RoboDK station: Config_3_New_Drillbit.rdk

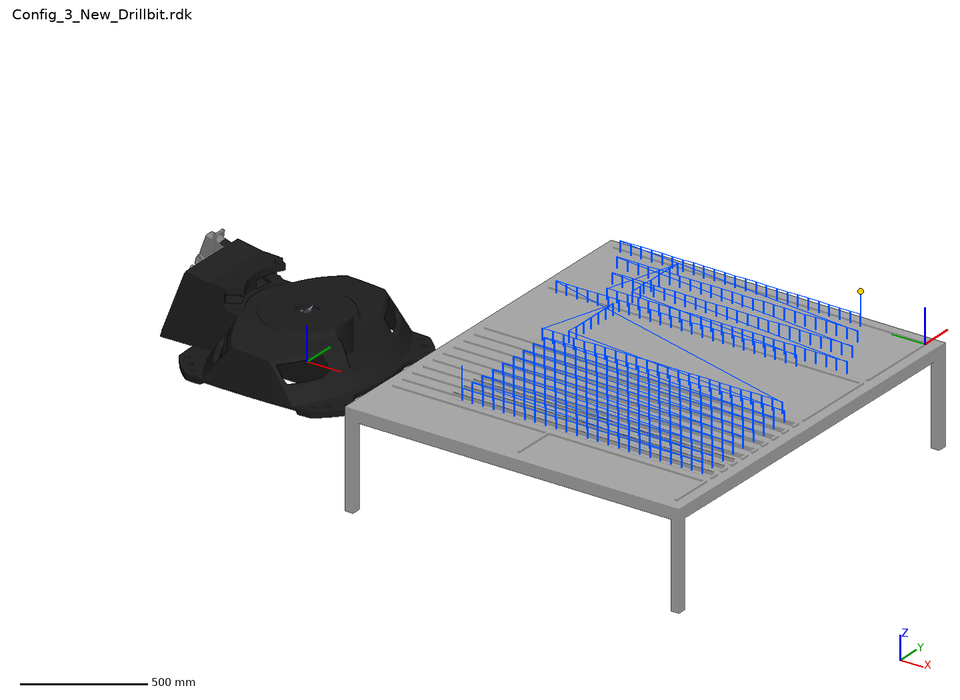
[picture v0: the station drawn from its stored meshes, robots at their saved joint values, targets as dots, program paths as lines]
Station Config_3_New_Drillbit (saved by RoboDK 5.2.3). Poses are relative to the parent item; angles as X-Y-Z fixed-axis rotations.
  - frame KUKA KR 210 R2700 extra Base at (0, 0, 0) mm
    - robot KUKA KR 210 R2700 extra: 6 axes, payload 210 kg, reach 2696 mm, repeatability 0.06 mm, weight 1068 kg
        joint limits [-185, -140, -120, -350, -125, -350] to [185, -5, 155, 350, 125, 350]; home [0, -90, 90, 0, 0, 0]; saved at [37.733, -88.827, 127.05, -51.844, 29.326, 78.997]
      - tool Spindle, TCP at (32, 0, 260) mm, rotated rx 0 ry 39 rz 0 deg, size 157.3 x 72 x 259.9 mm
  - frame Corner First Plate at (2495, 660, 510.8) mm, rotated rx 0 ry 0 rz 90 deg
  - object Table 3 at (1700, -800, 455) mm, rotated rx 0 ry 0 rz 90 deg, size 1820 x 1600 x 475 mm, geometry from Table 3.stl
  - object Config_3 at (2495, 660, 510.8) mm, rotated rx 0 ry 0 rz 90 deg
  - machining project Path1 settings: rotZ(0) | rotX(0)*rotY(0) | rotz(0) | onStart | onPathStart | onApproach | onPoint | onRetract | onFinish | SetRPM(%1) | SetTool(%1) | Extruder(%1) | default | default | OutOnMov(%1) | OutOffMov(%1) | onPathFinish | M_RunCode(%1)
  - program Path1 (1131 instructions, listed below)
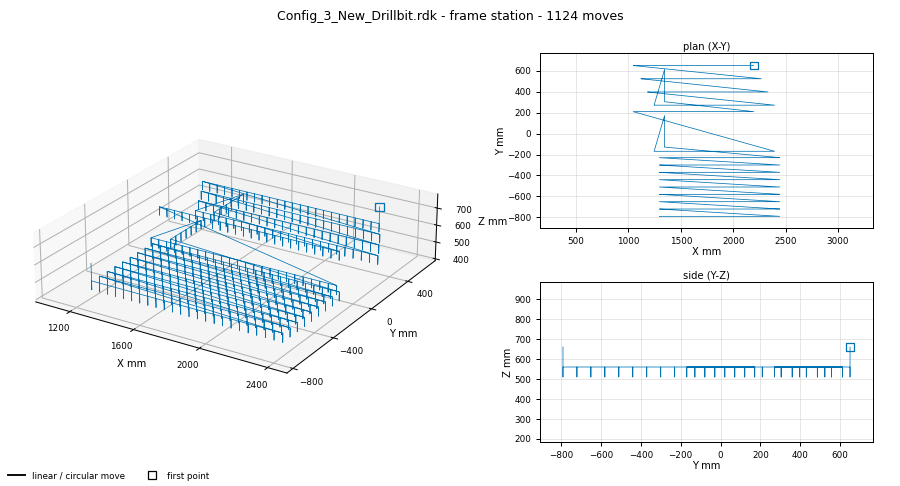
[picture p0: tool path of Config_3_New_Drillbit.rdk in frame station, 1124 of 1124 moves have a stored position in this frame; points joined in program order, loops and branches not executed]

--- program Path1 (robot KUKA KR 210 R2700 extra) ---
  Smooth(1)
  Set speed (1000.0 mm/s)
  Set Ref.: Corner First Plate
  Set Tool: Spindle
  Show Spindle
  MoveJ 1 to (-10.8, 300, 150) mm, rotated rx -180 ry 0 rz 90 deg; joints [-18.673, -56.771, 84.075, 25.785, 27.594, -37.894]
  MoveL 2 to (-10.8, 300, 150) mm, rotated rx -180 ry 0 rz 90 deg; joints [-18.673, -56.771, 84.075, 25.785, 27.594, -37.894]
  MoveL 3 to (-10.8, 300, 50) mm, rotated rx 180 ry 0 rz 90 deg; joints [-18.673, -54.184, 85.426, 29.563, 24.104, -42.09]
  MoveL 4 to (-10.8, 300, 50) mm, rotated rx 180 ry 0 rz 90 deg; joints [-18.673, -54.184, 85.426, 29.563, 24.104, -42.09]
  Set speed (150.0 mm/s)
  MoveL 5 to (-10.8, 300, -0.5) mm, rotated rx 180 ry 0 rz 90 deg; joints [-18.673, -52.769, 85.95, 31.865, 22.437, -44.595]
  MoveL 6 to (-10.8, 300, 50) mm, rotated rx 180 ry 0 rz 90 deg; joints [-18.673, -54.184, 85.426, 29.563, 24.104, -42.09]
  MoveL 7 to (-10.8, 350, 50) mm, rotated rx 180 ry 0 rz 90 deg; joints [-19.136, -56.141, 88.674, 31.59, 23.193, -44.569]
  MoveL 8 to (-10.8, 350, -0.5) mm, rotated rx 180 ry 0 rz 90 deg; joints [-19.136, -54.681, 89.197, 34.21, 21.527, -47.403]
  MoveL 9 to (-10.8, 350, 50) mm, rotated rx 180 ry 0 rz 90 deg; joints [-19.136, -56.141, 88.674, 31.59, 23.193, -44.569]
  MoveL 10 to (-10.8, 400, 50) mm, rotated rx -180 ry 0 rz 90 deg; joints [-19.622, -58.066, 91.821, 33.711, 22.382, -47.158]
  MoveL 11 to (-10.8, 400, -0.5) mm, rotated rx -180 ry 0 rz 90 deg; joints [-19.622, -56.557, 92.346, 36.679, 20.72, -50.348]
  MoveL 12 to (-10.8, 400, 50) mm, rotated rx -180 ry 0 rz 90 deg; joints [-19.622, -58.066, 91.821, 33.711, 22.382, -47.158]
  MoveL 13 to (-10.8, 450, 50) mm, rotated rx 180 ry 0 rz 90 deg; joints [-20.132, -59.962, 94.878, 35.915, 21.67, -49.846]
  MoveL 14 to (-10.8, 450, -0.5) mm, rotated rx -180 ry 0 rz 90 deg; joints [-20.132, -58.404, 95.405, 39.258, 20.016, -53.422]
  MoveL 15 to (-10.8, 450, 50) mm, rotated rx 180 ry 0 rz 90 deg; joints [-20.132, -59.962, 94.878, 35.915, 21.67, -49.846]
  MoveL 16 to (-10.8, 500, 50) mm, rotated rx 180 ry 0 rz 90 deg; joints [-20.668, -61.836, 97.851, 38.189, 21.056, -52.621]
  MoveL 17 to (-10.8, 500, -0.5) mm, rotated rx -180 ry 0 rz 90 deg; joints [-20.668, -60.227, 98.383, 41.928, 19.416, -56.606]
  MoveL 18 to (-10.8, 500, 50) mm, rotated rx 180 ry 0 rz 90 deg; joints [-20.668, -61.836, 97.851, 38.189, 21.056, -52.621]
  MoveL 19 to (-10.8, 550, 50) mm, rotated rx 180 ry 0 rz 90 deg; joints [-21.232, -63.693, 100.748, 40.512, 20.539, -55.465]
  MoveL 20 to (-10.8, 550, -0.5) mm, rotated rx -180 ry 0 rz 90 deg; joints [-21.232, -62.029, 101.285, 44.666, 18.917, -59.878]
  MoveL 21 to (-10.8, 550, 50) mm, rotated rx 180 ry 0 rz 90 deg; joints [-21.232, -63.693, 100.748, 40.512, 20.539, -55.465]
  MoveL 22 to (-10.8, 600, 50) mm, rotated rx -180 ry 0 rz 90 deg; joints [-21.826, -65.537, 103.573, 42.861, 20.119, -58.356]
  MoveL 23 to (-10.8, 600, -0.5) mm, rotated rx -180 ry 0 rz 90 deg; joints [-21.826, -63.817, 104.117, 47.441, 18.521, -63.209]
  MoveL 24 to (-10.8, 600, 50) mm, rotated rx -180 ry 0 rz 90 deg; joints [-21.826, -65.537, 103.573, 42.861, 20.119, -58.356]
  MoveL 25 to (-10.8, 650, 50) mm, rotated rx -180 ry 0 rz 90 deg; joints [-22.453, -67.372, 106.331, 45.208, 19.797, -61.269]
  MoveL 26 to (-10.8, 650, -0.5) mm, rotated rx 180 ry 0 rz 90 deg; joints [-22.453, -65.593, 106.883, 50.215, 18.227, -66.564]
  MoveL 27 to (-10.8, 650, 50) mm, rotated rx -180 ry 0 rz 90 deg; joints [-22.453, -67.372, 106.331, 45.208, 19.797, -61.269]
  MoveL 28 to (-10.8, 700, 50) mm, rotated rx -180 ry 0 rz 90 deg; joints [-23.115, -69.203, 109.025, 47.523, 19.571, -64.173]
  MoveL 29 to (-10.8, 700, -0.5) mm, rotated rx 180 ry 0 rz 90 deg; joints [-23.115, -67.362, 109.587, 52.95, 18.032, -69.905]
  MoveL 30 to (-10.8, 700, 50) mm, rotated rx -180 ry 0 rz 90 deg; joints [-23.115, -69.203, 109.025, 47.523, 19.571, -64.173]
  MoveL 31 to (-10.8, 750, 50) mm, rotated rx -180 ry 0 rz 90 deg; joints [-23.814, -71.033, 111.66, 49.773, 19.44, -67.039]
  MoveL 32 to (-10.8, 750, -0.5) mm, rotated rx 180 ry 0 rz 90 deg; joints [-23.814, -69.127, 112.233, 55.604, 17.936, -73.194]
  MoveL 33 to (-10.8, 750, 50) mm, rotated rx -180 ry 0 rz 90 deg; joints [-23.814, -71.033, 111.66, 49.773, 19.44, -67.039]
  MoveL 34 to (-10.8, 800, 50) mm, rotated rx -180 ry 0 rz 90 deg; joints [-24.555, -72.867, 114.238, 51.923, 19.404, -69.834]
  MoveL 35 to (-10.8, 800, -0.5) mm, rotated rx -180 ry 0 rz 90 deg; joints [-24.555, -70.893, 114.823, 58.134, 17.935, -76.388]
  MoveL 36 to (-10.8, 800, 50) mm, rotated rx -180 ry 0 rz 90 deg; joints [-24.555, -72.867, 114.238, 51.923, 19.404, -69.834]
  MoveL 37 to (-10.8, 850, 50) mm, rotated rx 180 ry 0 rz 90 deg; joints [-25.34, -74.708, 116.76, 53.942, 19.461, -72.529]
  MoveL 38 to (-10.8, 850, -0.5) mm, rotated rx -180 ry 0 rz 90 deg; joints [-25.34, -72.662, 117.358, 60.5, 18.027, -79.453]
  MoveL 39 to (-10.8, 850, 50) mm, rotated rx 180 ry 0 rz 90 deg; joints [-25.34, -74.708, 116.76, 53.942, 19.461, -72.529]
  MoveL 40 to (-10.8, 900, 50) mm, rotated rx -180 ry 0 rz 90 deg; joints [-26.173, -76.561, 119.228, 55.798, 19.61, -75.093]
  MoveL 41 to (-10.8, 900, -0.5) mm, rotated rx -180 ry 0 rz 90 deg; joints [-26.173, -74.439, 119.842, 62.666, 18.208, -82.352]
  MoveL 42 to (-10.8, 900, 50) mm, rotated rx -180 ry 0 rz 90 deg; joints [-26.173, -76.561, 119.228, 55.798, 19.61, -75.093]
  MoveL 43 to (-10.8, 950, 50) mm, rotated rx -180 ry 0 rz 90 deg; joints [-27.058, -78.43, 121.643, 57.462, 19.851, -77.502]
  MoveL 44 to (-10.8, 950, -0.5) mm, rotated rx 180 ry 0 rz 90 deg; joints [-27.058, -76.227, 122.274, 64.602, 18.476, -85.059]
  MoveL 45 to (-10.8, 950, 50) mm, rotated rx -180 ry 0 rz 90 deg; joints [-27.058, -78.43, 121.643, 57.462, 19.851, -77.502]
  MoveL 46 to (-10.8, 1000, 50) mm, rotated rx -180 ry 0 rz 90 deg; joints [-28.001, -80.318, 124.007, 58.912, 20.182, -79.735]
  MoveL 47 to (-10.8, 1000, -0.5) mm, rotated rx 180 ry 0 rz 90 deg; joints [-28.001, -78.031, 124.656, 66.28, 18.827, -87.549]
  MoveL 48 to (-10.8, 1000, 50) mm, rotated rx -180 ry 0 rz 90 deg; joints [-28.001, -80.318, 124.007, 58.912, 20.182, -79.735]
  MoveL 49 to (-10.8, 1050, 50) mm, rotated rx -180 ry 0 rz 90 deg; joints [-29.005, -82.231, 126.318, 60.129, 20.604, -81.776]
  MoveL 50 to (-10.8, 1050, -0.5) mm, rotated rx -180 ry 0 rz 90 deg; joints [-29.005, -79.854, 126.988, 67.681, 19.26, -89.808]
  MoveL 51 to (-10.8, 1050, 50) mm, rotated rx -180 ry 0 rz 90 deg; joints [-29.005, -82.231, 126.318, 60.129, 20.604, -81.776]
  MoveL 52 to (-10.8, 1100, 50) mm, rotated rx -180 ry 0 rz 90 deg; joints [-30.078, -84.172, 128.578, 61.097, 21.117, -83.613]
  MoveL 53 to (-10.8, 1100, -0.5) mm, rotated rx -180 ry 0 rz 90 deg; joints [-30.078, -81.701, 129.27, 68.792, 19.774, -91.823]
  MoveL 54 to (-10.8, 1100, 50) mm, rotated rx -180 ry 0 rz 90 deg; joints [-30.078, -84.172, 128.578, 61.097, 21.117, -83.613]
  MoveL 55 to (-10.8, 1150, 50) mm, rotated rx 180 ry 0 rz 90 deg; joints [-31.224, -86.147, 130.785, 61.808, 21.724, -85.24]
  MoveL 56 to (-10.8, 1150, -0.5) mm, rotated rx -180 ry 0 rz 90 deg; joints [-31.224, -83.576, 131.502, 69.603, 20.368, -93.59]
  MoveL 57 to (-10.8, 1150, 50) mm, rotated rx 180 ry 0 rz 90 deg; joints [-31.224, -86.147, 130.785, 61.808, 21.724, -85.24]
  MoveL 58 to (-10.8, 1200, 50) mm, rotated rx -180 ry 0 rz 90 deg; joints [-32.452, -88.16, 132.937, 62.257, 22.43, -86.657]
  MoveL 59 to (-10.8, 1200, -0.5) mm, rotated rx 180 ry 0 rz 90 deg; joints [-32.452, -85.485, 133.681, 70.11, 21.045, -95.109]
  MoveL 60 to (-10.8, 1200, 50) mm, rotated rx -180 ry 0 rz 90 deg; joints [-32.452, -88.16, 132.937, 62.257, 22.43, -86.657]
  MoveL 61 to (-10.8, 1250, 50) mm, rotated rx 180 ry 0 rz 90 deg; joints [-33.768, -90.216, 135.034, 62.444, 23.238, -87.866]
  MoveL 62 to (-10.8, 1250, -0.5) mm, rotated rx -180 ry 0 rz 90 deg; joints [-33.768, -87.431, 135.807, 70.315, 21.808, -96.384]
  MoveL 63 to (-10.8, 1250, 50) mm, rotated rx 180 ry 0 rz 90 deg; joints [-33.768, -90.216, 135.034, 62.444, 23.238, -87.866]
  MoveL 64 to (-10.8, 1300, 50) mm, rotated rx 180 ry 0 rz 90 deg; joints [-35.181, -92.32, 137.073, 62.376, 24.157, -88.879]
  MoveL 65 to (-10.8, 1300, -0.5) mm, rotated rx -180 ry 0 rz 90 deg; joints [-35.181, -89.419, 137.878, 70.222, 22.664, -97.425]
  MoveL 66 to (-10.8, 1300, 50) mm, rotated rx 180 ry 0 rz 90 deg; joints [-35.181, -92.32, 137.073, 62.376, 24.157, -88.879]
  MoveL 67 to (-10.8, 1350, 50) mm, rotated rx -180 ry 0 rz 90 deg; joints [-36.701, -94.476, 139.051, 62.061, 25.197, -89.708]
  MoveL 68 to (-10.8, 1350, -0.5) mm, rotated rx 180 ry 0 rz 90 deg; joints [-36.701, -91.455, 139.89, 69.839, 23.619, -98.245]
  MoveL 69 to (-10.8, 1350, 50) mm, rotated rx -180 ry 0 rz 90 deg; joints [-36.701, -94.476, 139.051, 62.061, 25.197, -89.708]
  MoveL 70 to (-10.8, 1400, 50) mm, rotated rx 180 ry 0 rz 90 deg; joints [-38.337, -96.689, 140.964, 61.514, 26.367, -90.372]
  MoveL 71 to (-10.8, 1400, -0.5) mm, rotated rx 180 ry 0 rz 90 deg; joints [-38.337, -93.543, 141.842, 69.179, 24.685, -98.863]
  MoveL 72 to (-10.8, 1400, 50) mm, rotated rx 180 ry 0 rz 90 deg; joints [-38.337, -96.689, 140.964, 61.514, 26.367, -90.372]
  MoveL 73 to (-10.8, 1450, 50) mm, rotated rx 180 ry 0 rz 90 deg; joints [-40.1, -98.961, 142.81, 60.755, 27.683, -90.897]
  MoveL 74 to (-10.8, 1450, -0.5) mm, rotated rx -180 ry 0 rz 90 deg; joints [-40.1, -95.687, 143.728, 68.26, 25.874, -99.3]
  MoveL 75 to (-10.8, 1450, 50) mm, rotated rx 180 ry 0 rz 90 deg; joints [-40.1, -98.961, 142.81, 60.755, 27.683, -90.897]
  MoveL 76 to (-136.94, 226.53, 50) mm, rotated rx -180 ry 0 rz 90 deg; joints [-14.696, -52.747, 83.017, 23.662, 23.44, -33.421]
  MoveL 77 to (-136.94, 226.53, -0.5) mm, rotated rx 180 ry 0 rz 90 deg; joints [-14.696, -51.366, 83.542, 25.573, 21.706, -35.49]
  MoveL 78 to (-136.94, 226.53, 50) mm, rotated rx -180 ry 0 rz 90 deg; joints [-14.696, -52.747, 83.017, 23.662, 23.44, -33.421]
  MoveL 79 to (-136.94, 276.53, 50) mm, rotated rx 180 ry 0 rz 90 deg; joints [-15.057, -54.772, 86.407, 25.489, 22.327, -35.605]
  MoveL 80 to (-136.94, 276.53, -0.5) mm, rotated rx -180 ry 0 rz 90 deg; joints [-15.057, -53.344, 86.931, 27.713, 20.582, -37.994]
  MoveL 81 to (-136.94, 276.53, 50) mm, rotated rx 180 ry 0 rz 90 deg; joints [-15.057, -54.772, 86.407, 25.489, 22.327, -35.605]
  MoveL 82 to (-136.94, 326.53, 50) mm, rotated rx 180 ry 0 rz 90 deg; joints [-15.435, -56.759, 89.689, 27.444, 21.31, -37.929]
  MoveL 83 to (-136.94, 326.53, -0.5) mm, rotated rx 180 ry 0 rz 90 deg; joints [-15.435, -55.284, 90.213, 30.025, 19.556, -40.683]
  MoveL 84 to (-136.94, 326.53, 50) mm, rotated rx 180 ry 0 rz 90 deg; joints [-15.435, -56.759, 89.689, 27.444, 21.31, -37.929]
  MoveL 85 to (-136.94, 376.53, 50) mm, rotated rx -180 ry 0 rz 90 deg; joints [-15.833, -58.716, 92.874, 29.528, 20.388, -40.394]
  MoveL 86 to (-136.94, 376.53, -0.5) mm, rotated rx 180 ry 0 rz 90 deg; joints [-15.833, -57.19, 93.4, 32.512, 18.63, -43.559]
  MoveL 87 to (-136.94, 376.53, 50) mm, rotated rx -180 ry 0 rz 90 deg; joints [-15.833, -58.716, 92.874, 29.528, 20.388, -40.394]
  MoveL 88 to (-136.94, 426.53, 50) mm, rotated rx 180 ry 0 rz 90 deg; joints [-16.251, -60.647, 95.97, 31.736, 19.561, -42.997]
  MoveL 89 to (-136.94, 426.53, -0.5) mm, rotated rx 180 ry 0 rz 90 deg; joints [-16.251, -59.071, 96.499, 35.17, 17.803, -46.621]
  MoveL 90 to (-136.94, 426.53, 50) mm, rotated rx 180 ry 0 rz 90 deg; joints [-16.251, -60.647, 95.97, 31.736, 19.561, -42.997]
  MoveL 91 to (-136.94, 476.53, 50) mm, rotated rx -180 ry 0 rz 90 deg; joints [-16.691, -62.56, 98.986, 34.06, 18.828, -45.731]
  MoveL 92 to (-136.94, 476.53, -0.5) mm, rotated rx -180 ry 0 rz 90 deg; joints [-16.691, -60.93, 99.52, 37.989, 17.077, -49.861]
  MoveL 93 to (-136.94, 476.53, 50) mm, rotated rx -180 ry 0 rz 90 deg; joints [-16.691, -62.56, 98.986, 34.06, 18.828, -45.731]
  MoveL 94 to (-136.94, 526.53, 50) mm, rotated rx 180 ry 0 rz 90 deg; joints [-17.155, -64.459, 101.928, 36.484, 18.191, -48.581]
  MoveL 95 to (-136.94, 526.53, -0.5) mm, rotated rx 180 ry 0 rz 90 deg; joints [-17.155, -62.773, 102.468, 40.951, 16.453, -53.259]
  MoveL 96 to (-136.94, 526.53, 50) mm, rotated rx 180 ry 0 rz 90 deg; joints [-17.155, -64.459, 101.928, 36.484, 18.191, -48.581]
  MoveL 97 to (-136.94, 576.53, 50) mm, rotated rx -180 ry 0 rz 90 deg; joints [-17.645, -66.35, 104.801, 38.987, 17.65, -51.528]
  MoveL 98 to (-136.94, 576.53, -0.5) mm, rotated rx 180 ry 0 rz 90 deg; joints [-17.645, -64.604, 105.349, 44.025, 15.931, -56.79]
  MoveL 99 to (-136.94, 576.53, 50) mm, rotated rx -180 ry 0 rz 90 deg; joints [-17.645, -66.35, 104.801, 38.987, 17.65, -51.528]
  MoveL 100 to (-136.94, 626.53, 50) mm, rotated rx -180 ry 0 rz 90 deg; joints [-18.163, -68.236, 107.61, 41.54, 17.206, -54.544]
  MoveL 101 to (-136.94, 626.53, -0.5) mm, rotated rx 180 ry 0 rz 90 deg; joints [-18.163, -66.429, 108.167, 47.173, 15.514, -60.415]
  MoveL 102 to (-136.94, 626.53, 50) mm, rotated rx -180 ry 0 rz 90 deg; joints [-18.163, -68.236, 107.61, 41.54, 17.206, -54.544]
  MoveL 103 to (-136.94, 676.53, 50) mm, rotated rx 180 ry 0 rz 90 deg; joints [-18.71, -70.124, 110.359, 44.108, 16.861, -57.597]
  MoveL 104 to (-136.94, 676.53, -0.5) mm, rotated rx 180 ry 0 rz 90 deg; joints [-18.71, -68.251, 110.926, 50.346, 15.201, -64.086]
  MoveL 105 to (-136.94, 676.53, 50) mm, rotated rx 180 ry 0 rz 90 deg; joints [-18.71, -70.124, 110.359, 44.108, 16.861, -57.597]
  MoveL 106 to (-136.94, 726.53, 50) mm, rotated rx -180 ry 0 rz 90 deg; joints [-19.291, -72.017, 113.051, 46.651, 16.613, -60.647]
  MoveL 107 to (-136.94, 726.53, -0.5) mm, rotated rx 180 ry 0 rz 90 deg; joints [-19.291, -70.075, 113.63, 53.486, 14.991, -67.75]
  MoveL 108 to (-136.94, 726.53, 50) mm, rotated rx -180 ry 0 rz 90 deg; joints [-19.291, -72.017, 113.051, 46.651, 16.613, -60.647]
  MoveL 109 to (-136.94, 776.53, 50) mm, rotated rx -180 ry 0 rz 90 deg; joints [-19.907, -73.921, 115.69, 49.122, 16.463, -63.65]
  MoveL 110 to (-136.94, 776.53, -0.5) mm, rotated rx -180 ry 0 rz 90 deg; joints [-19.907, -71.906, 116.282, 56.534, 14.884, -71.346]
  MoveL 111 to (-136.94, 776.53, 50) mm, rotated rx -180 ry 0 rz 90 deg; joints [-19.907, -73.921, 115.69, 49.122, 16.463, -63.65]
  MoveL 112 to (-136.94, 826.53, 50) mm, rotated rx -180 ry 0 rz 90 deg; joints [-20.562, -75.841, 118.277, 51.476, 16.411, -66.562]
  MoveL 113 to (-136.94, 826.53, -0.5) mm, rotated rx 180 ry 0 rz 90 deg; joints [-20.562, -73.748, 118.884, 59.426, 14.875, -74.816]
  MoveL 114 to (-136.94, 826.53, 50) mm, rotated rx -180 ry 0 rz 90 deg; joints [-20.562, -75.841, 118.277, 51.476, 16.411, -66.562]
  MoveL 115 to (-136.94, 876.53, 50) mm, rotated rx 180 ry 0 rz 90 deg; joints [-21.259, -77.781, 120.813, 53.664, 16.455, -69.337]
  MoveL 116 to (-136.94, 876.53, -0.5) mm, rotated rx 180 ry 0 rz 90 deg; joints [-21.259, -75.607, 121.438, 62.103, 14.963, -78.101]
  MoveL 117 to (-136.94, 876.53, 50) mm, rotated rx 180 ry 0 rz 90 deg; joints [-21.259, -77.781, 120.813, 53.664, 16.455, -69.337]
  MoveL 118 to (-136.94, 926.53, 50) mm, rotated rx 180 ry 0 rz 90 deg; joints [-22.003, -79.748, 123.302, 55.644, 16.595, -71.934]
  MoveL 119 to (-136.94, 926.53, -0.5) mm, rotated rx -180 ry 0 rz 90 deg; joints [-22.003, -77.487, 123.945, 64.512, 15.141, -81.151]
  MoveL 120 to (-136.94, 926.53, 50) mm, rotated rx 180 ry 0 rz 90 deg; joints [-22.003, -79.748, 123.302, 55.644, 16.595, -71.934]
  MoveL 121 to (-136.94, 976.53, 50) mm, rotated rx 180 ry 0 rz 90 deg; joints [-22.798, -81.747, 125.742, 57.374, 16.831, -74.315]
  MoveL 122 to (-136.94, 976.53, -0.5) mm, rotated rx 180 ry 0 rz 90 deg; joints [-22.798, -79.394, 126.407, 66.607, 15.408, -83.923]
  MoveL 123 to (-136.94, 976.53, 50) mm, rotated rx 180 ry 0 rz 90 deg; joints [-22.798, -81.747, 125.742, 57.374, 16.831, -74.315]
  MoveL 124 to (-136.94, 1026.53, 50) mm, rotated rx 180 ry 0 rz 90 deg; joints [-23.65, -83.786, 128.136, 58.822, 17.162, -76.449]
  MoveL 125 to (-136.94, 1026.53, -0.5) mm, rotated rx 180 ry 0 rz 90 deg; joints [-23.65, -81.334, 128.824, 68.353, 15.76, -86.384]
  MoveL 126 to (-136.94, 1026.53, 50) mm, rotated rx 180 ry 0 rz 90 deg; joints [-23.65, -83.786, 128.136, 58.822, 17.162, -76.449]
  MoveL 127 to (-136.94, 1076.53, 50) mm, rotated rx -180 ry 0 rz 90 deg; joints [-24.563, -85.871, 130.482, 59.961, 17.589, -78.313]
  MoveL 128 to (-136.94, 1076.53, -0.5) mm, rotated rx -180 ry 0 rz 90 deg; joints [-24.563, -83.315, 131.195, 69.722, 16.194, -88.511]
  MoveL 129 to (-136.94, 1076.53, 50) mm, rotated rx -180 ry 0 rz 90 deg; joints [-24.563, -85.871, 130.482, 59.961, 17.589, -78.313]
  MoveL 130 to (-136.94, 1126.53, 50) mm, rotated rx 180 ry 0 rz 90 deg; joints [-25.545, -88.01, 132.78, 60.772, 18.117, -79.89]
  MoveL 131 to (-136.94, 1126.53, -0.5) mm, rotated rx -180 ry 0 rz 90 deg; joints [-25.545, -85.343, 133.522, 70.696, 16.711, -90.288]
  MoveL 132 to (-136.94, 1126.53, 50) mm, rotated rx 180 ry 0 rz 90 deg; joints [-25.545, -88.01, 132.78, 60.772, 18.117, -79.89]
  MoveL 133 to (-136.94, 1176.53, 50) mm, rotated rx 180 ry 0 rz 90 deg; joints [-26.603, -90.212, 135.03, 61.243, 18.751, -81.173]
  MoveL 134 to (-136.94, 1176.53, -0.5) mm, rotated rx -180 ry 0 rz 90 deg; joints [-26.603, -87.427, 135.803, 71.264, 17.312, -91.708]
  MoveL 135 to (-136.94, 1176.53, 50) mm, rotated rx 180 ry 0 rz 90 deg; joints [-26.603, -90.212, 135.03, 61.243, 18.751, -81.173]
  MoveL 136 to (-136.94, 1226.53, 50) mm, rotated rx -180 ry 0 rz 90 deg; joints [-27.744, -92.486, 137.229, 61.372, 19.498, -82.16]
  MoveL 137 to (-136.94, 1226.53, -0.5) mm, rotated rx -180 ry 0 rz 90 deg; joints [-27.744, -89.576, 138.036, 71.423, 18.003, -92.77]
  MoveL 138 to (-136.94, 1226.53, 50) mm, rotated rx -180 ry 0 rz 90 deg; joints [-27.744, -92.486, 137.229, 61.372, 19.498, -82.16]
  MoveL 139 to (-136.94, 1276.53, 50) mm, rotated rx -180 ry 0 rz 90 deg; joints [-28.98, -94.842, 139.375, 61.162, 20.369, -82.86]
  MoveL 140 to (-136.94, 1276.53, -0.5) mm, rotated rx 180 ry 0 rz 90 deg; joints [-28.98, -91.801, 140.221, 71.174, 18.792, -93.483]
  MoveL 141 to (-136.94, 1276.53, 50) mm, rotated rx -180 ry 0 rz 90 deg; joints [-28.98, -94.842, 139.375, 61.162, 20.369, -82.86]
  MoveL 142 to (-136.94, 1326.53, 50) mm, rotated rx 180 ry 0 rz 90 deg; joints [-30.319, -97.292, 141.466, 60.624, 21.381, -83.287]
  MoveL 143 to (-136.94, 1326.53, -0.5) mm, rotated rx 180 ry 0 rz 90 deg; joints [-30.319, -94.113, 142.354, 70.527, 19.692, -93.857]
  MoveL 144 to (-136.94, 1326.53, 50) mm, rotated rx 180 ry 0 rz 90 deg; joints [-30.319, -97.292, 141.466, 60.624, 21.381, -83.287]
  MoveL 145 to (-136.94, 1376.53, 50) mm, rotated rx -180 ry 0 rz 90 deg; joints [-31.776, -99.848, 143.498, 59.78, 22.552, -83.466]
  MoveL 146 to (-136.94, 1376.53, -0.5) mm, rotated rx -180 ry 0 rz 90 deg; joints [-31.776, -96.524, 144.433, 69.496, 20.721, -93.913]
  MoveL 147 to (-136.94, 1376.53, 50) mm, rotated rx -180 ry 0 rz 90 deg; joints [-31.776, -99.848, 143.498, 59.78, 22.552, -83.466]
  MoveL 148 to (-263.08, 163.47, 50) mm, rotated rx -180 ry 0 rz 90 deg; joints [-10.919, -51.317, 80.596, 17.606, 23.211, -24.785]
  MoveL 149 to (-263.08, 163.47, -0.5) mm, rotated rx -180 ry 0 rz 90 deg; joints [-10.919, -49.967, 81.124, 19.044, 21.428, -26.34]
  MoveL 150 to (-263.08, 163.47, 50) mm, rotated rx -180 ry 0 rz 90 deg; joints [-10.919, -51.317, 80.596, 17.606, 23.211, -24.785]
  MoveL 151 to (-263.08, 213.47, 50) mm, rotated rx -180 ry 0 rz 90 deg; joints [-11.184, -53.402, 84.118, 19.086, 21.92, -26.532]
  MoveL 152 to (-263.08, 213.47, -0.5) mm, rotated rx 180 ry 0 rz 90 deg; joints [-11.184, -52.006, 84.643, 20.792, 20.113, -28.359]
  MoveL 153 to (-263.08, 213.47, 50) mm, rotated rx -180 ry 0 rz 90 deg; joints [-11.184, -53.402, 84.118, 19.086, 21.92, -26.532]
  MoveL 154 to (-263.08, 263.47, 50) mm, rotated rx -180 ry 0 rz 90 deg; joints [-11.463, -55.444, 87.522, 20.701, 20.719, -28.421]
  MoveL 155 to (-263.08, 263.47, -0.5) mm, rotated rx 180 ry 0 rz 90 deg; joints [-11.463, -54, 88.046, 22.723, 18.891, -30.569]
  MoveL 156 to (-263.08, 263.47, 50) mm, rotated rx -180 ry 0 rz 90 deg; joints [-11.463, -55.444, 87.522, 20.701, 20.719, -28.421]
  MoveL 157 to (-263.08, 313.47, 50) mm, rotated rx 180 ry 0 rz 90 deg; joints [-11.755, -57.451, 90.821, 22.46, 19.608, -30.463]
  MoveL 158 to (-263.08, 313.47, -0.5) mm, rotated rx -180 ry 0 rz 90 deg; joints [-11.755, -55.958, 91.346, 24.854, 17.76, -32.99]
  MoveL 159 to (-263.08, 313.47, 50) mm, rotated rx 180 ry 0 rz 90 deg; joints [-11.755, -57.451, 90.821, 22.46, 19.608, -30.463]
  MoveL 160 to (-263.08, 363.47, 50) mm, rotated rx -180 ry 0 rz 90 deg; joints [-12.062, -59.431, 94.026, 24.371, 18.585, -32.667]
  MoveL 161 to (-263.08, 363.47, -0.5) mm, rotated rx 180 ry 0 rz 90 deg; joints [-12.062, -57.887, 94.553, 27.202, 16.72, -35.637]
  MoveL 162 to (-263.08, 363.47, 50) mm, rotated rx -180 ry 0 rz 90 deg; joints [-12.062, -59.431, 94.026, 24.371, 18.585, -32.667]
  MoveL 163 to (-263.08, 413.47, 50) mm, rotated rx -180 ry 0 rz 90 deg; joints [-12.386, -61.389, 97.146, 26.438, 17.649, -35.037]
  MoveL 164 to (-263.08, 413.47, -0.5) mm, rotated rx 180 ry 0 rz 90 deg; joints [-12.386, -59.792, 97.676, 29.778, 15.771, -38.524]
  MoveL 165 to (-263.08, 413.47, 50) mm, rotated rx -180 ry 0 rz 90 deg; joints [-12.386, -61.389, 97.146, 26.438, 17.649, -35.037]
  MoveL 166 to (-263.08, 463.47, 50) mm, rotated rx 180 ry 0 rz 90 deg; joints [-12.727, -63.331, 100.187, 28.662, 16.801, -37.577]
  MoveL 167 to (-263.08, 463.47, -0.5) mm, rotated rx 180 ry 0 rz 90 deg; joints [-12.727, -61.678, 100.724, 32.588, 14.916, -41.658]
  MoveL 168 to (-263.08, 463.47, 50) mm, rotated rx 180 ry 0 rz 90 deg; joints [-12.727, -63.331, 100.187, 28.662, 16.801, -37.577]
  MoveL 169 to (-263.08, 513.47, 50) mm, rotated rx 180 ry 0 rz 90 deg; joints [-13.087, -65.264, 103.158, 31.038, 16.043, -40.283]
  MoveL 170 to (-263.08, 513.47, -0.5) mm, rotated rx 180 ry 0 rz 90 deg; joints [-13.087, -63.553, 103.701, 35.631, 14.158, -45.039]
  MoveL 171 to (-263.08, 513.47, 50) mm, rotated rx 180 ry 0 rz 90 deg; joints [-13.087, -65.264, 103.158, 31.038, 16.043, -40.283]
  MoveL 172 to (-263.08, 563.47, 50) mm, rotated rx -180 ry 0 rz 90 deg; joints [-13.467, -67.192, 106.063, 33.554, 15.377, -43.141]
  MoveL 173 to (-263.08, 563.47, -0.5) mm, rotated rx -180 ry 0 rz 90 deg; joints [-13.467, -65.419, 106.614, 38.891, 13.499, -48.652]
  MoveL 174 to (-263.08, 563.47, 50) mm, rotated rx -180 ry 0 rz 90 deg; joints [-13.467, -67.192, 106.063, 33.554, 15.377, -43.141]
  MoveL 175 to (-263.08, 613.47, 50) mm, rotated rx 180 ry 0 rz 90 deg; joints [-13.87, -69.121, 108.907, 36.187, 14.804, -46.133]
  MoveL 176 to (-263.08, 613.47, -0.5) mm, rotated rx 180 ry 0 rz 90 deg; joints [-13.87, -67.283, 109.468, 42.338, 12.944, -52.468]
  MoveL 177 to (-263.08, 613.47, 50) mm, rotated rx 180 ry 0 rz 90 deg; joints [-13.87, -69.121, 108.907, 36.187, 14.804, -46.133]
  MoveL 178 to (-263.08, 663.47, 50) mm, rotated rx -180 ry 0 rz 90 deg; joints [-14.297, -71.056, 111.693, 38.904, 14.328, -49.225]
  MoveL 179 to (-263.08, 663.47, -0.5) mm, rotated rx -180 ry 0 rz 90 deg; joints [-14.297, -69.15, 112.266, 45.923, 12.494, -56.44]
  MoveL 180 to (-263.08, 663.47, 50) mm, rotated rx -180 ry 0 rz 90 deg; joints [-14.297, -71.056, 111.693, 38.904, 14.328, -49.225]
  MoveL 181 to (-263.08, 713.47, 50) mm, rotated rx -180 ry 0 rz 90 deg; joints [-14.751, -73.003, 114.427, 41.662, 13.949, -52.376]
  MoveL 182 to (-263.08, 713.47, -0.5) mm, rotated rx 180 ry 0 rz 90 deg; joints [-14.751, -71.024, 115.012, 49.58, 12.15, -60.503]
  MoveL 183 to (-263.08, 713.47, 50) mm, rotated rx -180 ry 0 rz 90 deg; joints [-14.751, -73.003, 114.427, 41.662, 13.949, -52.376]
  MoveL 184 to (-263.08, 763.47, 50) mm, rotated rx -180 ry 0 rz 90 deg; joints [-15.234, -74.967, 117.109, 44.406, 13.67, -55.533]
  MoveL 185 to (-263.08, 763.47, -0.5) mm, rotated rx 180 ry 0 rz 90 deg; joints [-15.234, -72.911, 117.71, 53.225, 11.914, -64.575]
  MoveL 186 to (-263.08, 763.47, 50) mm, rotated rx -180 ry 0 rz 90 deg; joints [-15.234, -74.967, 117.109, 44.406, 13.67, -55.533]
  MoveL 187 to (-263.08, 813.47, 50) mm, rotated rx -180 ry 0 rz 90 deg; joints [-15.749, -76.955, 119.743, 47.073, 13.49, -58.634]
  MoveL 188 to (-263.08, 813.47, -0.5) mm, rotated rx -180 ry 0 rz 90 deg; joints [-15.749, -74.816, 120.361, 56.763, 11.784, -68.563]
  MoveL 189 to (-263.08, 813.47, 50) mm, rotated rx -180 ry 0 rz 90 deg; joints [-15.749, -76.955, 119.743, 47.073, 13.49, -58.634]
  MoveL 190 to (-263.08, 863.47, 50) mm, rotated rx 180 ry 0 rz 90 deg; joints [-16.299, -78.972, 122.331, 49.595, 13.411, -61.614]
  MoveL 191 to (-263.08, 863.47, -0.5) mm, rotated rx 180 ry 0 rz 90 deg; joints [-16.299, -76.746, 122.967, 60.097, 11.756, -72.371]
  MoveL 192 to (-263.08, 863.47, 50) mm, rotated rx 180 ry 0 rz 90 deg; joints [-16.299, -78.972, 122.331, 49.595, 13.411, -61.614]
  MoveL 193 to (-263.08, 913.47, 50) mm, rotated rx 180 ry 0 rz 90 deg; joints [-16.887, -81.027, 124.874, 51.903, 13.432, -64.404]
  MoveL 194 to (-263.08, 913.47, -0.5) mm, rotated rx -180 ry 0 rz 90 deg; joints [-16.887, -78.707, 125.531, 63.131, 11.826, -75.907]
  MoveL 195 to (-263.08, 913.47, 50) mm, rotated rx 180 ry 0 rz 90 deg; joints [-16.887, -81.027, 124.874, 51.903, 13.432, -64.404]
  MoveL 196 to (-263.08, 963.47, 50) mm, rotated rx 180 ry 0 rz 90 deg; joints [-17.518, -83.127, 127.373, 53.931, 13.554, -66.941]
  MoveL 197 to (-263.08, 963.47, -0.5) mm, rotated rx 180 ry 0 rz 90 deg; joints [-17.518, -80.708, 128.053, 65.783, 11.988, -79.089]
  MoveL 198 to (-263.08, 963.47, 50) mm, rotated rx 180 ry 0 rz 90 deg; joints [-17.518, -83.127, 127.373, 53.931, 13.554, -66.941]
  MoveL 199 to (-263.08, 1013.47, 50) mm, rotated rx 180 ry 0 rz 90 deg; joints [-18.197, -85.282, 129.829, 55.621, 13.776, -69.168]
  MoveL 200 to (-263.08, 1013.47, -0.5) mm, rotated rx 180 ry 0 rz 90 deg; joints [-18.197, -82.755, 130.535, 67.981, 12.239, -81.85]
  MoveL 201 to (-263.08, 1013.47, 50) mm, rotated rx 180 ry 0 rz 90 deg; joints [-18.197, -85.282, 129.829, 55.621, 13.776, -69.168]
  MoveL 202 to (-263.08, 1063.47, 50) mm, rotated rx 180 ry 0 rz 90 deg; joints [-18.928, -87.5, 132.242, 56.924, 14.1, -71.04]
  MoveL 203 to (-263.08, 1063.47, -0.5) mm, rotated rx -180 ry 0 rz 90 deg; joints [-18.928, -84.86, 132.977, 69.673, 12.574, -84.139]
  MoveL 204 to (-263.08, 1063.47, 50) mm, rotated rx 180 ry 0 rz 90 deg; joints [-18.928, -87.5, 132.242, 56.924, 14.1, -71.04]
  MoveL 205 to (-263.08, 1113.47, 50) mm, rotated rx -180 ry 0 rz 90 deg; joints [-19.718, -89.794, 134.612, 57.802, 14.532, -72.52]
  MoveL 206 to (-263.08, 1113.47, -0.5) mm, rotated rx 180 ry 0 rz 90 deg; joints [-19.718, -87.032, 135.379, 70.821, 12.991, -85.92]
  MoveL 207 to (-263.08, 1113.47, 50) mm, rotated rx -180 ry 0 rz 90 deg; joints [-19.718, -89.794, 134.612, 57.802, 14.532, -72.52]
  MoveL 208 to (-263.08, 1163.47, 50) mm, rotated rx 180 ry 0 rz 90 deg; joints [-20.574, -92.177, 136.938, 58.232, 15.077, -73.589]
  MoveL 209 to (-263.08, 1163.47, -0.5) mm, rotated rx 180 ry 0 rz 90 deg; joints [-20.574, -89.284, 137.74, 71.4, 13.494, -87.171]
  MoveL 210 to (-263.08, 1163.47, 50) mm, rotated rx 180 ry 0 rz 90 deg; joints [-20.574, -92.177, 136.938, 58.232, 15.077, -73.589]
  MoveL 211 to (-263.08, 1213.47, 50) mm, rotated rx -180 ry 0 rz 90 deg; joints [-21.503, -94.664, 139.218, 58.205, 15.748, -74.238]
  MoveL 212 to (-263.08, 1213.47, -0.5) mm, rotated rx 180 ry 0 rz 90 deg; joints [-21.503, -91.632, 140.06, 71.397, 14.087, -87.885]
  MoveL 213 to (-263.08, 1213.47, 50) mm, rotated rx -180 ry 0 rz 90 deg; joints [-21.503, -94.664, 139.218, 58.205, 15.748, -74.238]
  MoveL 214 to (-263.08, 1263.47, 50) mm, rotated rx 180 ry 0 rz 90 deg; joints [-22.516, -97.272, 141.45, 57.722, 16.562, -74.473]
  MoveL 215 to (-263.08, 1263.47, -0.5) mm, rotated rx 180 ry 0 rz 90 deg; joints [-22.516, -94.093, 142.337, 70.81, 14.784, -88.06]
  MoveL 216 to (-263.08, 1263.47, 50) mm, rotated rx 180 ry 0 rz 90 deg; joints [-22.516, -97.272, 141.45, 57.722, 16.562, -74.473]
  MoveL 217 to (-263.08, 1313.47, 50) mm, rotated rx -180 ry 0 rz 90 deg; joints [-23.624, -100.021, 143.63, 56.803, 17.54, -74.315]
  MoveL 218 to (-263.08, 1313.47, -0.5) mm, rotated rx -180 ry 0 rz 90 deg; joints [-23.624, -96.688, 144.568, 69.649, 15.604, -87.711]
  MoveL 219 to (-263.08, 1313.47, 50) mm, rotated rx -180 ry 0 rz 90 deg; joints [-23.624, -100.021, 143.63, 56.803, 17.54, -74.315]
  MoveL 220 to (-389.22, 100, 50) mm, rotated rx -180 ry 0 rz 90 deg; joints [-7.276, -49.461, 77.422, 11.443, 23.685, -16.168]
  MoveL 221 to (-389.22, 100, -0.5) mm, rotated rx -180 ry 0 rz 90 deg; joints [-7.276, -48.149, 77.954, 12.348, 21.881, -17.149]
  MoveL 222 to (-389.22, 100, 50) mm, rotated rx -180 ry 0 rz 90 deg; joints [-7.276, -49.461, 77.422, 11.443, 23.685, -16.168]
  MoveL 223 to (-389.22, 150, 50) mm, rotated rx 180 ry 0 rz 90 deg; joints [-7.449, -51.611, 81.094, 12.456, 22.228, -17.358]
  MoveL 224 to (-389.22, 150, -0.5) mm, rotated rx 180 ry 0 rz 90 deg; joints [-7.449, -50.254, 81.621, 13.542, 20.392, -18.524]
  MoveL 225 to (-389.22, 150, 50) mm, rotated rx 180 ry 0 rz 90 deg; joints [-7.449, -51.611, 81.094, 12.456, 22.228, -17.358]
  MoveL 226 to (-389.22, 200, 50) mm, rotated rx 180 ry 0 rz 90 deg; joints [-7.631, -53.71, 84.634, 13.574, 20.859, -18.659]
  MoveL 227 to (-389.22, 200, -0.5) mm, rotated rx 180 ry 0 rz 90 deg; joints [-7.631, -52.307, 85.158, 14.882, 18.991, -20.05]
  MoveL 228 to (-389.22, 200, 50) mm, rotated rx 180 ry 0 rz 90 deg; joints [-7.631, -53.71, 84.634, 13.574, 20.859, -18.659]
  MoveL 229 to (-389.22, 250, 50) mm, rotated rx 180 ry 0 rz 90 deg; joints [-7.823, -55.768, 88.058, 14.812, 19.575, -20.085]
  MoveL 230 to (-389.22, 250, -0.5) mm, rotated rx 180 ry 0 rz 90 deg; joints [-7.823, -54.316, 88.581, 16.389, 17.673, -21.748]
  MoveL 231 to (-389.22, 250, 50) mm, rotated rx 180 ry 0 rz 90 deg; joints [-7.823, -55.768, 88.058, 14.812, 19.575, -20.085]
  MoveL 232 to (-389.22, 300, 50) mm, rotated rx -180 ry 0 rz 90 deg; joints [-8.024, -57.793, 91.378, 16.182, 18.372, -21.649]
  MoveL 233 to (-389.22, 300, -0.5) mm, rotated rx 180 ry 0 rz 90 deg; joints [-8.024, -56.291, 91.902, 18.087, 16.436, -23.645]
  MoveL 234 to (-389.22, 300, 50) mm, rotated rx -180 ry 0 rz 90 deg; joints [-8.024, -57.793, 91.378, 16.182, 18.372, -21.649]
  MoveL 235 to (-389.22, 350, 50) mm, rotated rx 180 ry 0 rz 90 deg; joints [-8.235, -59.791, 94.605, 17.699, 17.248, -23.367]
  MoveL 236 to (-389.22, 350, -0.5) mm, rotated rx -180 ry 0 rz 90 deg; joints [-8.235, -58.238, 95.132, 20.004, 15.278, -25.768]
  MoveL 237 to (-389.22, 350, 50) mm, rotated rx 180 ry 0 rz 90 deg; joints [-8.235, -59.791, 94.605, 17.699, 17.248, -23.367]
  MoveL 238 to (-389.22, 400, 50) mm, rotated rx 180 ry 0 rz 90 deg; joints [-8.458, -61.771, 97.748, 19.375, 16.202, -25.252]
  MoveL 239 to (-389.22, 400, -0.5) mm, rotated rx 180 ry 0 rz 90 deg; joints [-8.458, -60.163, 98.28, 22.168, 14.201, -28.145]
  MoveL 240 to (-389.22, 400, 50) mm, rotated rx 180 ry 0 rz 90 deg; joints [-8.458, -61.771, 97.748, 19.375, 16.202, -25.252]
  MoveL 241 to (-389.22, 450, 50) mm, rotated rx -180 ry 0 rz 90 deg; joints [-8.693, -63.737, 100.815, 21.222, 15.234, -27.316]
  MoveL 242 to (-389.22, 450, -0.5) mm, rotated rx 180 ry 0 rz 90 deg; joints [-8.693, -62.072, 101.353, 24.607, 13.205, -30.807]
  MoveL 243 to (-389.22, 450, 50) mm, rotated rx -180 ry 0 rz 90 deg; joints [-8.693, -63.737, 100.815, 21.222, 15.234, -27.316]
  MoveL 244 to (-389.22, 500, 50) mm, rotated rx 180 ry 0 rz 90 deg; joints [-8.942, -65.695, 103.813, 23.25, 14.347, -29.571]
  MoveL 245 to (-389.22, 500, -0.5) mm, rotated rx -180 ry 0 rz 90 deg; joints [-8.942, -63.97, 104.358, 27.348, 12.294, -33.781]
  MoveL 246 to (-389.22, 500, 50) mm, rotated rx 180 ry 0 rz 90 deg; joints [-8.942, -65.695, 103.813, 23.25, 14.347, -29.571]
  MoveL 247 to (-389.22, 550, 50) mm, rotated rx 180 ry 0 rz 90 deg; joints [-9.205, -67.652, 106.747, 25.463, 13.542, -32.02]
  MoveL 248 to (-389.22, 550, -0.5) mm, rotated rx 180 ry 0 rz 90 deg; joints [-9.205, -65.864, 107.3, 30.411, 11.471, -37.087]
  MoveL 249 to (-389.22, 550, 50) mm, rotated rx 180 ry 0 rz 90 deg; joints [-9.205, -67.652, 106.747, 25.463, 13.542, -32.02]
  MoveL 250 to (-389.22, 600, 50) mm, rotated rx -180 ry 0 rz 90 deg; joints [-9.484, -69.613, 109.621, 27.857, 12.821, -34.66]
  MoveL 251 to (-389.22, 600, -0.5) mm, rotated rx 180 ry 0 rz 90 deg; joints [-9.484, -67.758, 110.185, 33.804, 10.741, -40.735]
  MoveL 252 to (-389.22, 600, 50) mm, rotated rx -180 ry 0 rz 90 deg; joints [-9.484, -69.613, 109.621, 27.857, 12.821, -34.66]
  MoveL 253 to (-389.22, 650, 50) mm, rotated rx 180 ry 0 rz 90 deg; joints [-9.78, -71.583, 112.44, 30.416, 12.19, -37.478]
  MoveL 254 to (-389.22, 650, -0.5) mm, rotated rx -180 ry 0 rz 90 deg; joints [-9.78, -69.657, 113.016, 37.514, 10.11, -44.711]
  MoveL 255 to (-389.22, 650, 50) mm, rotated rx 180 ry 0 rz 90 deg; joints [-9.78, -71.583, 112.44, 30.416, 12.19, -37.478]
  MoveL 256 to (-389.22, 700, 50) mm, rotated rx -180 ry 0 rz 90 deg; joints [-10.095, -73.57, 115.208, 33.111, 11.65, -40.445]
  MoveL 257 to (-389.22, 700, -0.5) mm, rotated rx -180 ry 0 rz 90 deg; joints [-10.095, -71.568, 115.798, 41.499, 9.583, -48.977]
  MoveL 258 to (-389.22, 700, 50) mm, rotated rx -180 ry 0 rz 90 deg; joints [-10.095, -73.57, 115.208, 33.111, 11.65, -40.445]
  MoveL 259 to (-389.22, 750, 50) mm, rotated rx -180 ry 0 rz 90 deg; joints [-10.431, -75.578, 117.928, 35.896, 11.205, -43.516]
  MoveL 260 to (-389.22, 750, -0.5) mm, rotated rx -180 ry 0 rz 90 deg; joints [-10.431, -73.497, 118.533, 45.682, 9.163, -53.456]
  MoveL 261 to (-389.22, 750, 50) mm, rotated rx -180 ry 0 rz 90 deg; joints [-10.431, -75.578, 117.928, 35.896, 11.205, -43.516]
  MoveL 262 to (-389.22, 800, 50) mm, rotated rx 180 ry 0 rz 90 deg; joints [-10.789, -77.616, 120.601, 38.705, 10.859, -46.625]
  MoveL 263 to (-389.22, 800, -0.5) mm, rotated rx -180 ry 0 rz 90 deg; joints [-10.789, -75.449, 121.225, 49.949, 8.853, -58.034]
  MoveL 264 to (-389.22, 800, 50) mm, rotated rx 180 ry 0 rz 90 deg; joints [-10.789, -77.616, 120.601, 38.705, 10.859, -46.625]
  MoveL 265 to (-389.22, 850, 50) mm, rotated rx -180 ry 0 rz 90 deg; joints [-11.173, -79.691, 123.231, 41.455, 10.614, -49.691]
  MoveL 266 to (-389.22, 850, -0.5) mm, rotated rx 180 ry 0 rz 90 deg; joints [-11.173, -77.432, 123.874, 54.149, 8.653, -62.564]
  MoveL 267 to (-389.22, 850, 50) mm, rotated rx -180 ry 0 rz 90 deg; joints [-11.173, -79.691, 123.231, 41.455, 10.614, -49.691]
  MoveL 268 to (-389.22, 900, 50) mm, rotated rx -180 ry 0 rz 90 deg; joints [-11.585, -81.811, 125.819, 44.048, 10.473, -52.619]
  MoveL 269 to (-389.22, 900, -0.5) mm, rotated rx 180 ry 0 rz 90 deg; joints [-11.585, -79.455, 126.484, 58.114, 8.559, -66.877]
  MoveL 270 to (-389.22, 900, 50) mm, rotated rx -180 ry 0 rz 90 deg; joints [-11.585, -81.811, 125.819, 44.048, 10.473, -52.619]
  MoveL 271 to (-389.22, 950, 50) mm, rotated rx 180 ry 0 rz 90 deg; joints [-12.027, -83.987, 128.366, 46.382, 10.436, -55.306]
  MoveL 272 to (-389.22, 950, -0.5) mm, rotated rx 180 ry 0 rz 90 deg; joints [-12.027, -81.525, 129.056, 61.672, 8.568, -70.804]
  MoveL 273 to (-389.22, 950, 50) mm, rotated rx 180 ry 0 rz 90 deg; joints [-12.027, -83.987, 128.366, 46.382, 10.436, -55.306]
  MoveL 274 to (-389.22, 1000, 50) mm, rotated rx 180 ry 0 rz 90 deg; joints [-12.505, -86.228, 130.873, 48.353, 10.507, -57.651]
  MoveL 275 to (-389.22, 1000, -0.5) mm, rotated rx -180 ry 0 rz 90 deg; joints [-12.505, -83.653, 131.591, 64.668, 8.671, -74.192]
  MoveL 276 to (-389.22, 1000, 50) mm, rotated rx 180 ry 0 rz 90 deg; joints [-12.505, -86.228, 130.873, 48.353, 10.507, -57.651]
  MoveL 277 to (-389.22, 1050, 50) mm, rotated rx 180 ry 0 rz 90 deg; joints [-13.021, -88.548, 133.341, 49.869, 10.687, -59.563]
  MoveL 278 to (-389.22, 1050, -0.5) mm, rotated rx -180 ry 0 rz 90 deg; joints [-13.021, -85.852, 134.09, 66.974, 8.862, -76.913]
  MoveL 279 to (-389.22, 1050, 50) mm, rotated rx 180 ry 0 rz 90 deg; joints [-13.021, -88.548, 133.341, 49.869, 10.687, -59.563]
  MoveL 280 to (-389.22, 1100, 50) mm, rotated rx 180 ry 0 rz 90 deg; joints [-13.58, -90.962, 135.769, 50.857, 10.984, -60.97]
  MoveL 281 to (-389.22, 1100, -0.5) mm, rotated rx -180 ry 0 rz 90 deg; joints [-13.58, -88.136, 136.553, 68.495, 9.139, -78.876]
  MoveL 282 to (-389.22, 1100, 50) mm, rotated rx 180 ry 0 rz 90 deg; joints [-13.58, -90.962, 135.769, 50.857, 10.984, -60.97]
  MoveL 283 to (-389.22, 1150, 50) mm, rotated rx 180 ry 0 rz 90 deg; joints [-14.189, -93.486, 138.156, 51.264, 11.406, -61.822]
  MoveL 284 to (-389.22, 1150, -0.5) mm, rotated rx 180 ry 0 rz 90 deg; joints [-14.189, -90.521, 138.98, 69.167, 9.5, -80.019]
  MoveL 285 to (-389.22, 1150, 50) mm, rotated rx 180 ry 0 rz 90 deg; joints [-14.189, -93.486, 138.156, 51.264, 11.406, -61.822]
  MoveL 286 to (-389.22, 1200, 50) mm, rotated rx -180 ry 0 rz 90 deg; joints [-14.854, -96.142, 140.502, 51.068, 11.97, -62.098]
  MoveL 287 to (-389.22, 1200, -0.5) mm, rotated rx 180 ry 0 rz 90 deg; joints [-14.854, -93.027, 141.37, 68.955, 9.954, -80.309]
  MoveL 288 to (-389.22, 1200, 50) mm, rotated rx -180 ry 0 rz 90 deg; joints [-14.854, -96.142, 140.502, 51.068, 11.97, -62.098]
  MoveL 289 to (-389.22, 1250, 50) mm, rotated rx -180 ry 0 rz 90 deg; joints [-15.583, -98.954, 142.804, 50.274, 12.698, -61.804]
  MoveL 290 to (-389.22, 1250, -0.5) mm, rotated rx -180 ry 0 rz 90 deg; joints [-15.583, -95.68, 143.722, 67.852, 10.517, -79.74]
  MoveL 291 to (-389.22, 1250, 50) mm, rotated rx -180 ry 0 rz 90 deg; joints [-15.583, -98.954, 142.804, 50.274, 12.698, -61.804]
  MoveL 292 to (-48.6, 1150, 50) mm, rotated rx -180 ry 0 rz 90 deg; joints [-29.722, -87.047, 131.759, 61.733, 20.748, -84.027]
  MoveL 293 to (-48.6, 1150, -0.5) mm, rotated rx 180 ry 0 rz 90 deg; joints [-29.722, -84.43, 132.488, 70.106, 19.379, -92.938]
  MoveL 294 to (-48.6, 1150, 50) mm, rotated rx -180 ry 0 rz 90 deg; joints [-29.722, -87.047, 131.759, 61.733, 20.748, -84.027]
  MoveL 295 to (-103.93, 1150, 50) mm, rotated rx -180 ry 0 rz 90 deg; joints [-27.44, -88.313, 133.097, 61.393, 19.289, -81.956]
  MoveL 296 to (-103.93, 1150, -0.5) mm, rotated rx 180 ry 0 rz 90 deg; joints [-27.44, -85.63, 133.842, 70.725, 17.892, -91.798]
  MoveL 297 to (-103.93, 1150, 50) mm, rotated rx -180 ry 0 rz 90 deg; joints [-27.44, -88.313, 133.097, 61.393, 19.289, -81.956]
  MoveL 298 to (-174.73, 1150, 50) mm, rotated rx 180 ry 0 rz 90 deg; joints [-24.376, -89.829, 134.647, 60.454, 17.371, -78.692]
  MoveL 299 to (-174.73, 1150, -0.5) mm, rotated rx -180 ry 0 rz 90 deg; joints [-24.376, -87.064, 135.414, 71.253, 15.92, -89.959]
  MoveL 300 to (-174.73, 1150, 50) mm, rotated rx 180 ry 0 rz 90 deg; joints [-24.376, -89.829, 134.647, 60.454, 17.371, -78.692]
  MoveL 301 to (-230.06, 1150, 50) mm, rotated rx 180 ry 0 rz 90 deg; joints [-21.873, -90.919, 135.727, 59.196, 15.841, -75.539]
  MoveL 302 to (-230.06, 1150, -0.5) mm, rotated rx 180 ry 0 rz 90 deg; joints [-21.873, -88.096, 136.511, 71.382, 14.324, -88.155]
  MoveL 303 to (-230.06, 1150, 50) mm, rotated rx 180 ry 0 rz 90 deg; joints [-21.873, -90.919, 135.727, 59.196, 15.841, -75.539]
  MoveL 304 to (-300.86, 1150, 50) mm, rotated rx 180 ry 0 rz 90 deg; joints [-18.539, -92.175, 136.935, 56.652, 13.859, -70.477]
  MoveL 305 to (-300.86, 1150, -0.5) mm, rotated rx -180 ry 0 rz 90 deg; joints [-18.539, -89.282, 137.738, 71.018, 12.216, -85.218]
  MoveL 306 to (-300.86, 1150, 50) mm, rotated rx 180 ry 0 rz 90 deg; joints [-18.539, -92.175, 136.935, 56.652, 13.859, -70.477]
  MoveL 307 to (-356.19, 1150, 50) mm, rotated rx -180 ry 0 rz 90 deg; joints [-15.838, -93.032, 137.738, 53.642, 12.314, -65.436]
  MoveL 308 to (-356.19, 1150, -0.5) mm, rotated rx 180 ry 0 rz 90 deg; joints [-15.838, -90.092, 138.554, 70.106, 10.524, -82.226]
  MoveL 309 to (-356.19, 1150, 50) mm, rotated rx -180 ry 0 rz 90 deg; joints [-15.838, -93.032, 137.738, 53.642, 12.314, -65.436]
  MoveL 310 to (-450.8, 300, 50) mm, rotated rx -180 ry 0 rz 90 deg; joints [-6.215, -58.102, 91.881, 12.873, 17.807, -17.113]
  MoveL 311 to (-450.8, 300, -0.5) mm, rotated rx 180 ry 0 rz 90 deg; joints [-6.215, -56.593, 92.406, 14.464, 15.83, -18.775]
  MoveL 312 to (-450.8, 300, 50) mm, rotated rx -180 ry 0 rz 90 deg; joints [-6.215, -58.102, 91.881, 12.873, 17.807, -17.113]
  MoveL 313 to (-450.8, 350, 50) mm, rotated rx 180 ry 0 rz 90 deg; joints [-6.38, -60.106, 95.108, 14.128, 16.649, -18.524]
  MoveL 314 to (-450.8, 350, -0.5) mm, rotated rx -180 ry 0 rz 90 deg; joints [-6.38, -58.544, 95.636, 16.073, 14.631, -20.543]
  MoveL 315 to (-450.8, 350, 50) mm, rotated rx 180 ry 0 rz 90 deg; joints [-6.38, -60.106, 95.108, 14.128, 16.649, -18.524]
  MoveL 316 to (-450.8, 400, 50) mm, rotated rx 180 ry 0 rz 90 deg; joints [-6.554, -62.091, 98.252, 15.527, 15.565, -20.085]
  MoveL 317 to (-450.8, 400, -0.5) mm, rotated rx 180 ry 0 rz 90 deg; joints [-6.554, -60.474, 98.784, 17.912, 13.506, -22.549]
  MoveL 318 to (-450.8, 400, 50) mm, rotated rx 180 ry 0 rz 90 deg; joints [-6.554, -62.091, 98.252, 15.527, 15.565, -20.085]
  MoveL 319 to (-450.8, 450, 50) mm, rotated rx 180 ry 0 rz 90 deg; joints [-6.737, -64.065, 101.321, 17.085, 14.554, -21.813]
  MoveL 320 to (-450.8, 450, -0.5) mm, rotated rx 180 ry 0 rz 90 deg; joints [-6.737, -62.39, 101.86, 20.018, 12.455, -24.828]
  MoveL 321 to (-450.8, 450, 50) mm, rotated rx 180 ry 0 rz 90 deg; joints [-6.737, -64.065, 101.321, 17.085, 14.554, -21.813]
  MoveL 322 to (-450.8, 500, 50) mm, rotated rx -180 ry 0 rz 90 deg; joints [-6.931, -66.032, 104.322, 18.817, 13.618, -23.721]
  MoveL 323 to (-450.8, 500, -0.5) mm, rotated rx 180 ry 0 rz 90 deg; joints [-6.931, -64.297, 104.869, 22.428, 11.481, -27.42]
  MoveL 324 to (-450.8, 500, 50) mm, rotated rx -180 ry 0 rz 90 deg; joints [-6.931, -66.032, 104.322, 18.817, 13.618, -23.721]
  MoveL 325 to (-450.8, 550, 50) mm, rotated rx 180 ry 0 rz 90 deg; joints [-7.136, -67.999, 107.26, 20.733, 12.758, -25.821]
  MoveL 326 to (-450.8, 550, -0.5) mm, rotated rx -180 ry 0 rz 90 deg; joints [-7.136, -66.2, 107.816, 25.181, 10.588, -30.361]
  MoveL 327 to (-450.8, 550, 50) mm, rotated rx 180 ry 0 rz 90 deg; joints [-7.136, -67.999, 107.26, 20.733, 12.758, -25.821]
  MoveL 328 to (-450.8, 600, 50) mm, rotated rx 180 ry 0 rz 90 deg; joints [-7.354, -69.972, 110.14, 22.839, 11.978, -28.119]
  MoveL 329 to (-450.8, 600, -0.5) mm, rotated rx -180 ry 0 rz 90 deg; joints [-7.354, -68.105, 110.707, 28.308, 9.78, -33.687]
  MoveL 330 to (-450.8, 600, 50) mm, rotated rx 180 ry 0 rz 90 deg; joints [-7.354, -69.972, 110.14, 22.839, 11.978, -28.119]
  MoveL 331 to (-450.8, 650, 50) mm, rotated rx -180 ry 0 rz 90 deg; joints [-7.585, -71.957, 112.966, 25.131, 11.28, -30.612]
  MoveL 332 to (-450.8, 650, -0.5) mm, rotated rx 180 ry 0 rz 90 deg; joints [-7.585, -70.017, 113.545, 31.829, 9.063, -37.416]
  MoveL 333 to (-450.8, 650, 50) mm, rotated rx -180 ry 0 rz 90 deg; joints [-7.585, -71.957, 112.966, 25.131, 11.28, -30.612]
  MoveL 334 to (-450.8, 700, 50) mm, rotated rx 180 ry 0 rz 90 deg; joints [-7.832, -73.959, 115.742, 27.592, 10.67, -33.285]
  MoveL 335 to (-450.8, 700, -0.5) mm, rotated rx -180 ry 0 rz 90 deg; joints [-7.832, -71.943, 116.335, 35.736, 8.443, -41.542]
  MoveL 336 to (-450.8, 700, 50) mm, rotated rx 180 ry 0 rz 90 deg; joints [-7.832, -73.959, 115.742, 27.592, 10.67, -33.285]
  MoveL 337 to (-450.8, 750, 50) mm, rotated rx -180 ry 0 rz 90 deg; joints [-8.094, -75.987, 118.47, 30.188, 10.15, -36.103]
  MoveL 338 to (-450.8, 750, -0.5) mm, rotated rx -180 ry 0 rz 90 deg; joints [-8.094, -73.888, 119.079, 39.985, 7.926, -46.022]
  MoveL 339 to (-450.8, 750, 50) mm, rotated rx -180 ry 0 rz 90 deg; joints [-8.094, -75.987, 118.47, 30.188, 10.15, -36.103]
  MoveL 340 to (-450.8, 800, 50) mm, rotated rx -180 ry 0 rz 90 deg; joints [-8.375, -78.046, 121.154, 32.862, 9.726, -39.012]
  MoveL 341 to (-450.8, 800, -0.5) mm, rotated rx 180 ry 0 rz 90 deg; joints [-8.375, -75.86, 121.781, 44.477, 7.518, -50.757]
  MoveL 342 to (-450.8, 800, 50) mm, rotated rx -180 ry 0 rz 90 deg; joints [-8.375, -78.046, 121.154, 32.862, 9.726, -39.012]
  MoveL 343 to (-450.8, 850, 50) mm, rotated rx 180 ry 0 rz 90 deg; joints [-8.676, -80.146, 123.795, 35.535, 9.401, -41.932]
  MoveL 344 to (-450.8, 850, -0.5) mm, rotated rx -180 ry 0 rz 90 deg; joints [-8.676, -77.867, 124.442, 49.054, 7.22, -55.591]
  MoveL 345 to (-450.8, 850, 50) mm, rotated rx 180 ry 0 rz 90 deg; joints [-8.676, -80.146, 123.795, 35.535, 9.401, -41.932]
  MoveL 346 to (-450.8, 900, 50) mm, rotated rx 180 ry 0 rz 90 deg; joints [-8.999, -82.295, 126.395, 38.103, 9.179, -44.761]
  MoveL 347 to (-450.8, 900, -0.5) mm, rotated rx 180 ry 0 rz 90 deg; joints [-8.999, -79.915, 127.066, 53.508, 7.033, -60.317]
  MoveL 348 to (-450.8, 900, 50) mm, rotated rx 180 ry 0 rz 90 deg; joints [-8.999, -82.295, 126.395, 38.103, 9.179, -44.761]
  MoveL 349 to (-450.8, 950, 50) mm, rotated rx -180 ry 0 rz 90 deg; joints [-9.347, -84.504, 128.955, 40.447, 9.065, -47.382]
  MoveL 350 to (-450.8, 950, -0.5) mm, rotated rx -180 ry 0 rz 90 deg; joints [-9.347, -82.017, 129.652, 57.6, 6.953, -64.698]
  MoveL 351 to (-450.8, 950, 50) mm, rotated rx -180 ry 0 rz 90 deg; joints [-9.347, -84.504, 128.955, 40.447, 9.065, -47.382]
  MoveL 352 to (-450.8, 1000, 50) mm, rotated rx 180 ry 0 rz 90 deg; joints [-9.723, -86.785, 131.477, 42.441, 9.061, -49.668]
  MoveL 353 to (-450.8, 1000, -0.5) mm, rotated rx -180 ry 0 rz 90 deg; joints [-9.723, -84.181, 132.203, 61.093, 6.973, -68.497]
  MoveL 354 to (-450.8, 1000, 50) mm, rotated rx 180 ry 0 rz 90 deg; joints [-9.723, -86.785, 131.477, 42.441, 9.061, -49.668]
  MoveL 355 to (-450.8, 1050, 50) mm, rotated rx 180 ry 0 rz 90 deg; joints [-10.13, -89.151, 133.961, 43.967, 9.174, -51.503]
  MoveL 356 to (-450.8, 1050, -0.5) mm, rotated rx -180 ry 0 rz 90 deg; joints [-10.13, -86.423, 134.719, 63.779, 7.087, -71.509]
  MoveL 357 to (-450.8, 1050, 50) mm, rotated rx 180 ry 0 rz 90 deg; joints [-10.13, -89.151, 133.961, 43.967, 9.174, -51.503]
  MoveL 358 to (-450.8, 1100, 50) mm, rotated rx -180 ry 0 rz 90 deg; joints [-10.571, -91.62, 136.406, 44.925, 9.41, -52.789]
  MoveL 359 to (-450.8, 1100, -0.5) mm, rotated rx 180 ry 0 rz 90 deg; joints [-10.571, -88.758, 137.2, 65.501, 7.289, -73.577]
  MoveL 360 to (-450.8, 1100, 50) mm, rotated rx -180 ry 0 rz 90 deg; joints [-10.571, -91.62, 136.406, 44.925, 9.41, -52.789]
  MoveL 361 to (-450.8, 1150, 50) mm, rotated rx -180 ry 0 rz 90 deg; joints [-11.053, -94.21, 138.812, 45.246, 9.782, -53.459]
  MoveL 362 to (-450.8, 1150, -0.5) mm, rotated rx -180 ry 0 rz 90 deg; joints [-11.053, -91.204, 139.648, 66.152, 7.58, -74.597]
  MoveL 363 to (-450.8, 1150, 50) mm, rotated rx -180 ry 0 rz 90 deg; joints [-11.053, -94.21, 138.812, 45.246, 9.782, -53.459]
  MoveL 364 to (-450.8, 1200, 50) mm, rotated rx -180 ry 0 rz 90 deg; joints [-11.58, -96.945, 141.178, 44.903, 10.309, -53.485]
  MoveL 365 to (-450.8, 1200, -0.5) mm, rotated rx -180 ry 0 rz 90 deg; joints [-11.58, -93.785, 142.06, 65.678, 7.969, -74.517]
  MoveL 366 to (-450.8, 1200, 50) mm, rotated rx -180 ry 0 rz 90 deg; joints [-11.58, -96.945, 141.178, 44.903, 10.309, -53.485]
  MoveL 367 to (-450.8, 1250, 50) mm, rotated rx -180 ry 0 rz 90 deg; joints [-12.159, -99.852, 143.501, 43.912, 11.018, -52.885]
  MoveL 368 to (-450.8, 1250, -0.5) mm, rotated rx -180 ry 0 rz 90 deg; joints [-12.159, -96.528, 144.436, 64.079, 8.475, -73.337]
  MoveL 369 to (-450.8, 1250, 50) mm, rotated rx -180 ry 0 rz 90 deg; joints [-12.159, -99.852, 143.501, 43.912, 11.018, -52.885]
  MoveL 370 to (-450.8, 1300, 50) mm, rotated rx -180 ry 0 rz 90 deg; joints [-12.798, -102.966, 145.779, 42.33, 11.948, -51.718]
  MoveL 371 to (-450.8, 1300, -0.5) mm, rotated rx -180 ry 0 rz 90 deg; joints [-12.798, -99.47, 146.773, 61.412, 9.135, -71.116]
  MoveL 372 to (-450.8, 1300, 50) mm, rotated rx -180 ry 0 rz 90 deg; joints [-12.798, -102.966, 145.779, 42.33, 11.948, -51.718]
  MoveL 373 to (-450.8, 1350, 50) mm, rotated rx -180 ry 0 rz 90 deg; joints [-13.507, -106.329, 148.005, 40.257, 13.147, -50.082]
  MoveL 374 to (-450.8, 1350, -0.5) mm, rotated rx -180 ry 0 rz 90 deg; joints [-13.507, -102.653, 149.068, 57.804, 10.002, -67.98]
  MoveL 375 to (-450.8, 1350, 50) mm, rotated rx -180 ry 0 rz 90 deg; joints [-13.507, -106.329, 148.005, 40.257, 13.147, -50.082]
  MoveL 376 to (-450.8, 1400, 50) mm, rotated rx 180 ry 0 rz 90 deg; joints [-14.296, -109.989, 150.175, 37.819, 14.681, -48.104]
  MoveL 377 to (-450.8, 1400, -0.5) mm, rotated rx -180 ry 0 rz 90 deg; joints [-14.296, -106.134, 151.316, 53.454, 11.153, -64.132]
  MoveL 378 to (-450.8, 1400, 50) mm, rotated rx 180 ry 0 rz 90 deg; joints [-14.296, -109.989, 150.175, 37.819, 14.681, -48.104]
  MoveL 379 to (-450.8, 1450, 50) mm, rotated rx 180 ry 0 rz 90 deg; joints [-15.182, -114.009, 152.278, 35.161, 16.63, -45.925]
  MoveL 380 to (-450.8, 1450, -0.5) mm, rotated rx 180 ry 0 rz 90 deg; joints [-15.182, -109.981, 153.51, 48.629, 12.687, -59.834]
  MoveL 381 to (-450.8, 1450, 50) mm, rotated rx 180 ry 0 rz 90 deg; joints [-15.182, -114.009, 152.278, 35.161, 16.63, -45.925]
  MoveL 382 to (-829.2, 100, 50) mm, rotated rx 180 ry 0 rz 90 deg; joints [4.561, -49.92, 78.21, -7.368, 22.969, 10.337]
  MoveL 383 to (-829.2, 100, -0.5) mm, rotated rx 180 ry 0 rz 90 deg; joints [4.561, -48.599, 78.741, -7.979, 21.134, 10.996]
  MoveL 384 to (-829.2, 100, 50) mm, rotated rx 180 ry 0 rz 90 deg; joints [4.561, -49.92, 78.21, -7.368, 22.969, 10.337]
  MoveL 385 to (-829.2, 150, 50) mm, rotated rx 180 ry 0 rz 90 deg; joints [4.671, -52.069, 81.871, -8.044, 21.484, 11.124]
  MoveL 386 to (-829.2, 150, -0.5) mm, rotated rx 180 ry 0 rz 90 deg; joints [4.671, -50.702, 82.397, -8.783, 19.611, 11.913]
  MoveL 387 to (-829.2, 150, 50) mm, rotated rx 180 ry 0 rz 90 deg; joints [4.671, -52.069, 81.871, -8.044, 21.484, 11.124]
  MoveL 388 to (-829.2, 200, 50) mm, rotated rx 180 ry 0 rz 90 deg; joints [4.786, -54.17, 85.403, -8.796, 20.082, 11.991]
  MoveL 389 to (-829.2, 200, -0.5) mm, rotated rx 180 ry 0 rz 90 deg; joints [4.786, -52.756, 85.927, -9.694, 18.169, 12.941]
  MoveL 390 to (-829.2, 200, 50) mm, rotated rx 180 ry 0 rz 90 deg; joints [4.786, -54.17, 85.403, -8.796, 20.082, 11.991]
  MoveL 391 to (-829.2, 250, 50) mm, rotated rx 180 ry 0 rz 90 deg; joints [4.907, -56.231, 88.821, -9.635, 18.759, 12.949]
  MoveL 392 to (-829.2, 250, -0.5) mm, rotated rx -180 ry 0 rz 90 deg; joints [4.907, -54.768, 89.345, -10.731, 16.804, 14.099]
  MoveL 393 to (-829.2, 250, 50) mm, rotated rx 180 ry 0 rz 90 deg; joints [4.907, -56.231, 88.821, -9.635, 18.759, 12.949]
  MoveL 394 to (-829.2, 300, 50) mm, rotated rx -180 ry 0 rz 90 deg; joints [5.034, -58.261, 92.139, -10.575, 17.51, 14.011]
  MoveL 395 to (-829.2, 300, -0.5) mm, rotated rx 180 ry 0 rz 90 deg; joints [5.034, -56.748, 92.664, -11.916, 15.511, 15.41]
  MoveL 396 to (-829.2, 300, 50) mm, rotated rx -180 ry 0 rz 90 deg; joints [5.034, -58.261, 92.139, -10.575, 17.51, 14.011]
  MoveL 397 to (-829.2, 350, 50) mm, rotated rx 180 ry 0 rz 90 deg; joints [5.168, -60.267, 95.365, -11.627, 16.334, 15.19]
  MoveL 398 to (-829.2, 350, -0.5) mm, rotated rx 180 ry 0 rz 90 deg; joints [5.168, -58.701, 95.893, -13.277, 14.288, 16.901]
  MoveL 399 to (-829.2, 350, 50) mm, rotated rx 180 ry 0 rz 90 deg; joints [5.168, -60.267, 95.365, -11.627, 16.334, 15.19]
  MoveL 400 to (-829.2, 400, 50) mm, rotated rx -180 ry 0 rz 90 deg; joints [5.309, -62.256, 98.51, -12.807, 15.228, 16.502]
  MoveL 401 to (-829.2, 400, -0.5) mm, rotated rx -180 ry 0 rz 90 deg; joints [5.309, -60.634, 99.043, -14.845, 13.136, 18.604]
  MoveL 402 to (-829.2, 400, 50) mm, rotated rx -180 ry 0 rz 90 deg; joints [5.309, -62.256, 98.51, -12.807, 15.228, 16.502]
  MoveL 403 to (-829.2, 450, 50) mm, rotated rx 180 ry 0 rz 90 deg; joints [5.458, -64.233, 101.581, -14.13, 14.192, 17.962]
  MoveL 404 to (-829.2, 450, -0.5) mm, rotated rx 180 ry 0 rz 90 deg; joints [5.458, -62.553, 102.12, -16.657, 12.053, 20.556]
  MoveL 405 to (-829.2, 450, 50) mm, rotated rx 180 ry 0 rz 90 deg; joints [5.458, -64.233, 101.581, -14.13, 14.192, 17.962]
  MoveL 406 to (-829.2, 500, 50) mm, rotated rx 180 ry 0 rz 90 deg; joints [5.615, -66.205, 104.584, -15.611, 13.228, 19.585]
  MoveL 407 to (-829.2, 500, -0.5) mm, rotated rx 180 ry 0 rz 90 deg; joints [5.615, -64.464, 105.131, -18.755, 11.041, 22.801]
  MoveL 408 to (-829.2, 500, 50) mm, rotated rx 180 ry 0 rz 90 deg; joints [5.615, -66.205, 104.584, -15.611, 13.228, 19.585]
  MoveL 409 to (-829.2, 550, 50) mm, rotated rx -180 ry 0 rz 90 deg; joints [5.782, -68.178, 107.524, -17.262, 12.336, 21.386]
  MoveL 410 to (-829.2, 550, -0.5) mm, rotated rx 180 ry 0 rz 90 deg; joints [5.782, -66.372, 108.08, -21.184, 10.105, 25.383]
  MoveL 411 to (-829.2, 550, 50) mm, rotated rx -180 ry 0 rz 90 deg; joints [5.782, -68.178, 107.524, -17.262, 12.336, 21.386]
  MoveL 412 to (-829.2, 600, 50) mm, rotated rx -180 ry 0 rz 90 deg; joints [5.959, -70.157, 110.407, -19.096, 11.52, 23.376]
  MoveL 413 to (-829.2, 600, -0.5) mm, rotated rx 180 ry 0 rz 90 deg; joints [5.959, -68.283, 110.974, -23.99, 9.247, 28.351]
  MoveL 414 to (-829.2, 600, 50) mm, rotated rx -180 ry 0 rz 90 deg; joints [5.959, -70.157, 110.407, -19.096, 11.52, 23.376]
  MoveL 415 to (-829.2, 650, 50) mm, rotated rx 180 ry 0 rz 90 deg; joints [6.147, -72.149, 113.236, -21.114, 10.783, 25.558]
  MoveL 416 to (-829.2, 650, -0.5) mm, rotated rx 180 ry 0 rz 90 deg; joints [6.147, -70.202, 113.816, -27.215, 8.474, 31.745]
  MoveL 417 to (-829.2, 650, 50) mm, rotated rx 180 ry 0 rz 90 deg; joints [6.147, -72.149, 113.236, -21.114, 10.783, 25.558]
  MoveL 418 to (-829.2, 700, 50) mm, rotated rx -180 ry 0 rz 90 deg; joints [6.348, -74.16, 116.016, -23.309, 10.128, 27.925]
  MoveL 419 to (-829.2, 700, -0.5) mm, rotated rx -180 ry 0 rz 90 deg; joints [6.348, -72.136, 116.611, -30.882, 7.791, 35.59]
  MoveL 420 to (-829.2, 700, 50) mm, rotated rx -180 ry 0 rz 90 deg; joints [6.348, -74.16, 116.016, -23.309, 10.128, 27.925]
  MoveL 421 to (-829.2, 750, 50) mm, rotated rx 180 ry 0 rz 90 deg; joints [6.562, -76.197, 118.749, -25.659, 9.56, 30.456]
  MoveL 422 to (-829.2, 750, -0.5) mm, rotated rx 180 ry 0 rz 90 deg; joints [6.562, -74.09, 119.36, -34.982, 7.206, 39.877]
  MoveL 423 to (-829.2, 750, 50) mm, rotated rx 180 ry 0 rz 90 deg; joints [6.562, -76.197, 118.749, -25.659, 9.56, 30.456]
  MoveL 424 to (-829.2, 800, 50) mm, rotated rx 180 ry 0 rz 90 deg; joints [6.791, -78.268, 121.438, -28.117, 9.085, 33.104]
  MoveL 425 to (-829.2, 800, -0.5) mm, rotated rx 180 ry 0 rz 90 deg; joints [6.791, -76.073, 122.067, -39.45, 6.725, 44.543]
  MoveL 426 to (-829.2, 800, 50) mm, rotated rx 180 ry 0 rz 90 deg; joints [6.791, -78.268, 121.438, -28.117, 9.085, 33.104]
  MoveL 427 to (-829.2, 850, 50) mm, rotated rx 180 ry 0 rz 90 deg; joints [7.036, -80.381, 124.084, -30.612, 8.707, 35.801]
  MoveL 428 to (-829.2, 850, -0.5) mm, rotated rx 180 ry 0 rz 90 deg; joints [7.036, -78.091, 124.735, -44.151, 6.354, 49.453]
  MoveL 429 to (-829.2, 850, 50) mm, rotated rx 180 ry 0 rz 90 deg; joints [7.036, -80.381, 124.084, -30.612, 8.707, 35.801]
  MoveL 430 to (-829.2, 900, 50) mm, rotated rx -180 ry 0 rz 90 deg; joints [7.299, -82.546, 126.691, -33.047, 8.431, 38.448]
  MoveL 431 to (-829.2, 900, -0.5) mm, rotated rx -180 ry 0 rz 90 deg; joints [7.299, -80.154, 127.364, -48.867, 6.094, 54.391]
  MoveL 432 to (-829.2, 900, 50) mm, rotated rx -180 ry 0 rz 90 deg; joints [7.299, -82.546, 126.691, -33.047, 8.431, 38.448]
  MoveL 433 to (-829.2, 950, 50) mm, rotated rx 180 ry 0 rz 90 deg; joints [7.583, -84.772, 129.258, -35.298, 8.263, 40.924]
  MoveL 434 to (-829.2, 950, -0.5) mm, rotated rx -180 ry 0 rz 90 deg; joints [7.583, -82.271, 129.958, -53.317, 5.944, 59.075]
  MoveL 435 to (-829.2, 950, 50) mm, rotated rx 180 ry 0 rz 90 deg; joints [7.583, -84.772, 129.258, -35.298, 8.263, 40.924]
  MoveL 436 to (-829.2, 1000, 50) mm, rotated rx -180 ry 0 rz 90 deg; joints [7.89, -87.074, 131.788, -37.231, 8.209, 43.094]
  MoveL 437 to (-829.2, 1000, -0.5) mm, rotated rx 180 ry 0 rz 90 deg; joints [7.89, -84.456, 132.517, -57.189, 5.9, 63.198]
  MoveL 438 to (-829.2, 1000, 50) mm, rotated rx -180 ry 0 rz 90 deg; joints [7.89, -87.074, 131.788, -37.231, 8.209, 43.094]
  MoveL 439 to (-829.2, 1050, 50) mm, rotated rx 180 ry 0 rz 90 deg; joints [8.222, -89.465, 134.28, -38.71, 8.274, 44.825]
  MoveL 440 to (-829.2, 1050, -0.5) mm, rotated rx 180 ry 0 rz 90 deg; joints [8.222, -86.72, 135.042, -60.194, 5.954, 66.468]
  MoveL 441 to (-829.2, 1050, 50) mm, rotated rx 180 ry 0 rz 90 deg; joints [8.222, -89.465, 134.28, -38.71, 8.274, 44.825]
  MoveL 442 to (-829.2, 1100, 50) mm, rotated rx 180 ry 0 rz 90 deg; joints [8.584, -91.963, 136.734, -39.62, 8.47, 46.002]
  MoveL 443 to (-829.2, 1100, -0.5) mm, rotated rx 180 ry 0 rz 90 deg; joints [8.584, -89.082, 137.534, -62.098, 6.101, 68.654]
  MoveL 444 to (-829.2, 1100, 50) mm, rotated rx 180 ry 0 rz 90 deg; joints [8.584, -91.963, 136.734, -39.62, 8.47, 46.002]
  MoveL 445 to (-829.2, 1150, 50) mm, rotated rx -180 ry 0 rz 90 deg; joints [8.978, -94.588, 139.15, -39.881, 8.81, 46.547]
  MoveL 446 to (-829.2, 1150, -0.5) mm, rotated rx 180 ry 0 rz 90 deg; joints [8.978, -91.561, 139.992, -62.744, 6.343, 69.6]
  MoveL 447 to (-829.2, 1150, 50) mm, rotated rx -180 ry 0 rz 90 deg; joints [8.978, -94.588, 139.15, -39.881, 8.81, 46.547]
  MoveL 448 to (-829.2, 1200, 50) mm, rotated rx 180 ry 0 rz 90 deg; joints [9.41, -97.365, 141.527, -39.465, 9.316, 46.431]
  MoveL 449 to (-829.2, 1200, -0.5) mm, rotated rx 180 ry 0 rz 90 deg; joints [9.41, -94.182, 142.416, -62.059, 6.688, 69.236]
  MoveL 450 to (-829.2, 1200, 50) mm, rotated rx 180 ry 0 rz 90 deg; joints [9.41, -97.365, 141.527, -39.465, 9.316, 46.431]
  MoveL 451 to (-829.2, 1250, 50) mm, rotated rx 180 ry 0 rz 90 deg; joints [9.885, -100.325, 143.861, -38.395, 10.018, 45.68]
  MoveL 452 to (-829.2, 1250, -0.5) mm, rotated rx 180 ry 0 rz 90 deg; joints [9.885, -96.975, 144.804, -60.059, 7.162, 67.577]
  MoveL 453 to (-829.2, 1250, 50) mm, rotated rx 180 ry 0 rz 90 deg; joints [9.885, -100.325, 143.861, -38.395, 10.018, 45.68]
  MoveL 454 to (-488.6, 1150, 50) mm, rotated rx -180 ry 0 rz 90 deg; joints [-9.093, -94.569, 139.134, 40.212, 8.861, -46.963]
  MoveL 455 to (-488.6, 1150, -0.5) mm, rotated rx -180 ry 0 rz 90 deg; joints [-9.093, -91.543, 139.975, 62.975, 6.41, -69.919]
  MoveL 456 to (-488.6, 1150, 50) mm, rotated rx -180 ry 0 rz 90 deg; joints [-9.093, -94.569, 139.134, 40.212, 8.861, -46.963]
  MoveL 457 to (-538.6, 1150, 50) mm, rotated rx 180 ry 0 rz 90 deg; joints [-6.467, -94.94, 139.462, 31.508, 7.795, -36.306]
  MoveL 458 to (-538.6, 1150, -0.5) mm, rotated rx -180 ry 0 rz 90 deg; joints [-6.467, -91.893, 140.309, 55.85, 4.914, -60.786]
  MoveL 459 to (-538.6, 1150, 50) mm, rotated rx 180 ry 0 rz 90 deg; joints [-6.467, -94.94, 139.462, 31.508, 7.795, -36.306]
  MoveL 460 to (-588.6, 1150, 50) mm, rotated rx 180 ry 0 rz 90 deg; joints [-3.814, -95.188, 139.679, 20.111, 6.993, -22.939]
  MoveL 461 to (-588.6, 1150, -0.5) mm, rotated rx 180 ry 0 rz 90 deg; joints [-3.814, -92.127, 140.53, 42.092, 3.581, -45.002]
  MoveL 462 to (-588.6, 1150, 50) mm, rotated rx 180 ry 0 rz 90 deg; joints [-3.814, -95.188, 139.679, 20.111, 6.993, -22.939]
  MoveL 463 to (-638.6, 1150, 50) mm, rotated rx -180 ry 0 rz 90 deg; joints [-1.145, -95.307, 139.783, 6.31, 6.569, -7.158]
  MoveL 464 to (-638.6, 1150, -0.5) mm, rotated rx 180 ry 0 rz 90 deg; joints [-1.145, -92.24, 140.637, 15.444, 2.706, -16.317]
  MoveL 465 to (-638.6, 1150, 50) mm, rotated rx -180 ry 0 rz 90 deg; joints [-1.145, -95.307, 139.783, 6.31, 6.569, -7.158]
  MoveL 466 to (-688.6, 1150, 50) mm, rotated rx 180 ry 0 rz 90 deg; joints [1.53, -95.298, 139.775, -8.401, 6.603, 9.535]
  MoveL 467 to (-688.6, 1150, -0.5) mm, rotated rx -180 ry 0 rz 90 deg; joints [1.53, -92.231, 140.629, -20.236, 2.784, 21.403]
  MoveL 468 to (-688.6, 1150, 50) mm, rotated rx 180 ry 0 rz 90 deg; joints [1.53, -95.298, 139.775, -8.401, 6.603, 9.535]
  MoveL 469 to (-738.6, 1150, 50) mm, rotated rx -180 ry 0 rz 90 deg; joints [4.198, -95.16, 139.654, -21.919, 7.088, 25.032]
  MoveL 470 to (-738.6, 1150, -0.5) mm, rotated rx -180 ry 0 rz 90 deg; joints [4.198, -92.1, 140.505, -44.706, 3.754, 47.909]
  MoveL 471 to (-738.6, 1150, 50) mm, rotated rx -180 ry 0 rz 90 deg; joints [4.198, -95.16, 139.654, -21.919, 7.088, 25.032]
  MoveL 472 to (-788.6, 1150, 50) mm, rotated rx 180 ry 0 rz 90 deg; joints [6.847, -94.894, 139.421, -32.922, 7.935, 38.002]
  MoveL 473 to (-788.6, 1150, -0.5) mm, rotated rx -180 ry 0 rz 90 deg; joints [6.847, -91.85, 140.268, -57.171, 5.123, 62.397]
  MoveL 474 to (-788.6, 1150, 50) mm, rotated rx 180 ry 0 rz 90 deg; joints [6.847, -94.894, 139.421, -32.922, 7.935, 38.002]
  MoveL 475 to (-890, 50, 50) mm, rotated rx 180 ry 0 rz 90 deg; joints [6.048, -47.46, 73.966, -9.052, 24.924, 12.928]
  MoveL 476 to (-890, 50, -0.5) mm, rotated rx -180 ry 0 rz 90 deg; joints [6.048, -46.189, 74.505, -9.714, 23.138, 13.653]
  MoveL 477 to (-890, 50, 50) mm, rotated rx 180 ry 0 rz 90 deg; joints [6.048, -47.46, 73.966, -9.052, 24.924, 12.928]
  MoveL 478 to (-890, 100, 50) mm, rotated rx 180 ry 0 rz 90 deg; joints [6.189, -49.67, 77.782, -9.853, 23.36, 13.876]
  MoveL 479 to (-890, 100, -0.5) mm, rotated rx 180 ry 0 rz 90 deg; joints [6.189, -48.355, 78.314, -10.648, 21.542, 14.737]
  MoveL 480 to (-890, 100, 50) mm, rotated rx 180 ry 0 rz 90 deg; joints [6.189, -49.67, 77.782, -9.853, 23.36, 13.876]
  MoveL 481 to (-890, 150, 50) mm, rotated rx -180 ry 0 rz 90 deg; joints [6.337, -51.82, 81.449, -10.738, 21.89, 14.913]
  MoveL 482 to (-890, 150, -0.5) mm, rotated rx 180 ry 0 rz 90 deg; joints [6.337, -50.459, 81.976, -11.697, 20.038, 15.939]
  MoveL 483 to (-890, 150, 50) mm, rotated rx -180 ry 0 rz 90 deg; joints [6.337, -51.82, 81.449, -10.738, 21.89, 14.913]
  MoveL 484 to (-890, 200, 50) mm, rotated rx 180 ry 0 rz 90 deg; joints [6.493, -53.92, 84.986, -11.72, 20.508, 16.05]
  MoveL 485 to (-890, 200, -0.5) mm, rotated rx 180 ry 0 rz 90 deg; joints [6.493, -52.512, 85.51, -12.878, 18.619, 17.28]
  MoveL 486 to (-890, 200, 50) mm, rotated rx 180 ry 0 rz 90 deg; joints [6.493, -53.92, 84.986, -11.72, 20.508, 16.05]
  MoveL 487 to (-890, 250, 50) mm, rotated rx -180 ry 0 rz 90 deg; joints [6.656, -55.979, 88.407, -12.811, 19.206, 17.301]
  MoveL 488 to (-890, 250, -0.5) mm, rotated rx 180 ry 0 rz 90 deg; joints [6.656, -54.523, 88.93, -14.215, 17.281, 18.779]
  MoveL 489 to (-890, 250, 50) mm, rotated rx -180 ry 0 rz 90 deg; joints [6.656, -55.979, 88.407, -12.811, 19.206, 17.301]
  MoveL 490 to (-890, 300, 50) mm, rotated rx 180 ry 0 rz 90 deg; joints [6.828, -58.007, 91.725, -14.024, 17.983, 18.68]
  MoveL 491 to (-890, 300, -0.5) mm, rotated rx 180 ry 0 rz 90 deg; joints [6.828, -56.5, 92.25, -15.73, 16.02, 20.464]
  MoveL 492 to (-890, 300, 50) mm, rotated rx 180 ry 0 rz 90 deg; joints [6.828, -58.007, 91.725, -14.024, 17.983, 18.68]
  MoveL 493 to (-890, 350, 50) mm, rotated rx -180 ry 0 rz 90 deg; joints [7.008, -60.009, 94.952, -15.373, 16.836, 20.201]
  MoveL 494 to (-890, 350, -0.5) mm, rotated rx -180 ry 0 rz 90 deg; joints [7.008, -58.449, 95.48, -17.453, 14.834, 22.362]
  MoveL 495 to (-890, 350, 50) mm, rotated rx -180 ry 0 rz 90 deg; joints [7.008, -60.009, 94.952, -15.373, 16.836, 20.201]
  MoveL 496 to (-890, 400, 50) mm, rotated rx 180 ry 0 rz 90 deg; joints [7.199, -61.992, 98.096, -16.874, 15.764, 21.88]
  MoveL 497 to (-890, 400, -0.5) mm, rotated rx -180 ry 0 rz 90 deg; joints [7.199, -60.378, 98.628, -19.414, 13.724, 24.506]
  MoveL 498 to (-890, 400, 50) mm, rotated rx 180 ry 0 rz 90 deg; joints [7.199, -61.992, 98.096, -16.874, 15.764, 21.88]
  MoveL 499 to (-890, 450, 50) mm, rotated rx 180 ry 0 rz 90 deg; joints [7.4, -63.963, 101.165, -18.54, 14.768, 23.731]
  MoveL 500 to (-890, 450, -0.5) mm, rotated rx -180 ry 0 rz 90 deg; joints [7.4, -62.292, 101.703, -21.649, 12.692, 26.93]
  MoveL 501 to (-890, 450, 50) mm, rotated rx 180 ry 0 rz 90 deg; joints [7.4, -63.963, 101.165, -18.54, 14.768, 23.731]
  MoveL 502 to (-890, 500, 50) mm, rotated rx -180 ry 0 rz 90 deg; joints [7.612, -65.928, 104.165, -20.385, 13.847, 25.769]
  MoveL 503 to (-890, 500, -0.5) mm, rotated rx 180 ry 0 rz 90 deg; joints [7.612, -64.196, 104.711, -24.19, 11.739, 29.671]
  MoveL 504 to (-890, 500, 50) mm, rotated rx -180 ry 0 rz 90 deg; joints [7.612, -65.928, 104.165, -20.385, 13.847, 25.769]
  MoveL 505 to (-890, 550, 50) mm, rotated rx -180 ry 0 rz 90 deg; joints [7.837, -67.892, 107.102, -22.415, 13.006, 28.001]
  MoveL 506 to (-890, 550, -0.5) mm, rotated rx -180 ry 0 rz 90 deg; joints [7.837, -66.096, 107.656, -27.072, 10.869, 32.759]
  MoveL 507 to (-890, 550, 50) mm, rotated rx -180 ry 0 rz 90 deg; joints [7.837, -67.892, 107.102, -22.415, 13.006, 28.001]
  MoveL 508 to (-890, 600, 50) mm, rotated rx 180 ry 0 rz 90 deg; joints [8.076, -69.861, 109.98, -24.635, 12.245, 30.432]
  MoveL 509 to (-890, 600, -0.5) mm, rotated rx -180 ry 0 rz 90 deg; joints [8.076, -67.997, 110.545, -30.316, 10.087, 36.221]
  MoveL 510 to (-890, 600, 50) mm, rotated rx 180 ry 0 rz 90 deg; joints [8.076, -69.861, 109.98, -24.635, 12.245, 30.432]
  MoveL 511 to (-890, 650, 50) mm, rotated rx -180 ry 0 rz 90 deg; joints [8.329, -71.841, 112.804, -27.037, 11.57, 33.055]
  MoveL 512 to (-890, 650, -0.5) mm, rotated rx -180 ry 0 rz 90 deg; joints [8.329, -69.906, 113.382, -33.932, 9.4, 40.065]
  MoveL 513 to (-890, 650, 50) mm, rotated rx -180 ry 0 rz 90 deg; joints [8.329, -71.841, 112.804, -27.037, 11.57, 33.055]
  MoveL 514 to (-890, 700, 50) mm, rotated rx 180 ry 0 rz 90 deg; joints [8.599, -73.838, 115.577, -29.598, 10.983, 35.848]
  MoveL 515 to (-890, 700, -0.5) mm, rotated rx 180 ry 0 rz 90 deg; joints [8.599, -71.827, 116.169, -37.897, 8.812, 44.271]
  MoveL 516 to (-890, 700, 50) mm, rotated rx 180 ry 0 rz 90 deg; joints [8.599, -73.838, 115.577, -29.598, 10.983, 35.848]
  MoveL 517 to (-890, 750, 50) mm, rotated rx 180 ry 0 rz 90 deg; joints [8.887, -75.86, 118.302, -32.281, 10.488, 38.775]
  MoveL 518 to (-890, 750, -0.5) mm, rotated rx -180 ry 0 rz 90 deg; joints [8.887, -73.767, 118.91, -42.154, 8.329, 48.78]
  MoveL 519 to (-890, 750, 50) mm, rotated rx 180 ry 0 rz 90 deg; joints [8.887, -75.86, 118.302, -32.281, 10.488, 38.775]
  MoveL 520 to (-890, 800, 50) mm, rotated rx -180 ry 0 rz 90 deg; joints [9.194, -77.913, 120.983, -35.023, 10.091, 41.774]
  MoveL 521 to (-890, 800, -0.5) mm, rotated rx 180 ry 0 rz 90 deg; joints [9.194, -75.733, 121.609, -46.593, 7.956, 53.486]
  MoveL 522 to (-890, 800, 50) mm, rotated rx -180 ry 0 rz 90 deg; joints [9.194, -77.913, 120.983, -35.023, 10.091, 41.774]
  MoveL 523 to (-890, 850, 50) mm, rotated rx 180 ry 0 rz 90 deg; joints [9.524, -80.005, 123.62, -37.744, 9.794, 44.766]
  MoveL 524 to (-890, 850, -0.5) mm, rotated rx 180 ry 0 rz 90 deg; joints [9.524, -77.732, 124.267, -51.056, 7.694, 58.231]
  MoveL 525 to (-890, 850, 50) mm, rotated rx 180 ry 0 rz 90 deg; joints [9.524, -80.005, 123.62, -37.744, 9.794, 44.766]
  MoveL 526 to (-890, 900, 50) mm, rotated rx -180 ry 0 rz 90 deg; joints [9.877, -82.145, 126.217, -40.339, 9.6, 47.647]
  MoveL 527 to (-890, 900, -0.5) mm, rotated rx 180 ry 0 rz 90 deg; joints [9.877, -79.772, 126.886, -55.347, 7.541, 62.82]
  MoveL 528 to (-890, 900, 50) mm, rotated rx -180 ry 0 rz 90 deg; joints [9.877, -82.145, 126.217, -40.339, 9.6, 47.647]
  MoveL 529 to (-890, 950, 50) mm, rotated rx 180 ry 0 rz 90 deg; joints [10.258, -84.343, 128.773, -42.695, 9.513, 50.306]
  MoveL 530 to (-890, 950, -0.5) mm, rotated rx -180 ry 0 rz 90 deg; joints [10.258, -81.864, 129.467, -59.25, 7.493, 67.04]
  MoveL 531 to (-890, 950, 50) mm, rotated rx 180 ry 0 rz 90 deg; joints [10.258, -84.343, 128.773, -42.695, 9.513, 50.306]
  MoveL 532 to (-890, 1000, 50) mm, rotated rx -180 ry 0 rz 90 deg; joints [10.668, -86.612, 131.29, -44.693, 9.535, 52.624]
  MoveL 533 to (-890, 1000, -0.5) mm, rotated rx 180 ry 0 rz 90 deg; joints [10.668, -84.017, 132.013, -62.561, 7.543, 70.686]
  MoveL 534 to (-890, 1000, 50) mm, rotated rx -180 ry 0 rz 90 deg; joints [10.668, -86.612, 131.29, -44.693, 9.535, 52.624]
  MoveL 535 to (-890, 1050, 50) mm, rotated rx 180 ry 0 rz 90 deg; joints [11.113, -88.964, 133.769, -46.223, 9.671, 54.493]
  MoveL 536 to (-890, 1050, -0.5) mm, rotated rx -180 ry 0 rz 90 deg; joints [11.113, -86.246, 134.524, -65.104, 7.685, 73.586]
  MoveL 537 to (-890, 1050, 50) mm, rotated rx 180 ry 0 rz 90 deg; joints [11.113, -88.964, 133.769, -46.223, 9.671, 54.493]
  MoveL 538 to (-890, 1100, 50) mm, rotated rx 180 ry 0 rz 90 deg; joints [11.595, -91.415, 136.209, -47.195, 9.928, 55.824]
  MoveL 539 to (-890, 1100, -0.5) mm, rotated rx -180 ry 0 rz 90 deg; joints [11.595, -88.564, 137, -66.748, 7.913, 75.609]
  MoveL 540 to (-890, 1100, 50) mm, rotated rx 180 ry 0 rz 90 deg; joints [11.595, -91.415, 136.209, -47.195, 9.928, 55.824]
  MoveL 541 to (-890, 1150, 50) mm, rotated rx 180 ry 0 rz 90 deg; joints [12.121, -93.984, 138.609, -47.547, 10.317, 56.557]
  MoveL 542 to (-890, 1150, -0.5) mm, rotated rx -180 ry 0 rz 90 deg; joints [12.121, -90.991, 139.441, -67.405, 8.229, 76.669]
  MoveL 543 to (-890, 1150, 50) mm, rotated rx 180 ry 0 rz 90 deg; joints [12.121, -93.984, 138.609, -47.547, 10.317, 56.557]
  MoveL 544 to (-890, 1200, 50) mm, rotated rx -180 ry 0 rz 90 deg; joints [12.696, -96.694, 140.969, -47.251, 10.856, 56.665]
  MoveL 545 to (-890, 1200, -0.5) mm, rotated rx -180 ry 0 rz 90 deg; joints [12.696, -93.548, 141.846, -67.028, 8.64, 76.722]
  MoveL 546 to (-890, 1200, 50) mm, rotated rx -180 ry 0 rz 90 deg; joints [12.696, -96.694, 140.969, -47.251, 10.856, 56.665]
  MoveL 547 to (-960, 50, 50) mm, rotated rx 180 ry 0 rz 90 deg; joints [7.868, -47.076, 73.298, -11.545, 25.494, 16.577]
  MoveL 548 to (-960, 50, -0.5) mm, rotated rx 180 ry 0 rz 90 deg; joints [7.868, -45.813, 73.839, -12.361, 23.73, 17.474]
  MoveL 549 to (-960, 50, 50) mm, rotated rx 180 ry 0 rz 90 deg; joints [7.868, -47.076, 73.298, -11.545, 25.494, 16.577]
  MoveL 550 to (-960, 100, 50) mm, rotated rx 180 ry 0 rz 90 deg; joints [8.051, -49.289, 77.128, -12.541, 23.948, 17.764]
  MoveL 551 to (-960, 100, -0.5) mm, rotated rx 180 ry 0 rz 90 deg; joints [8.051, -47.982, 77.66, -13.516, 22.155, 18.824]
  MoveL 552 to (-960, 100, 50) mm, rotated rx 180 ry 0 rz 90 deg; joints [8.051, -49.289, 77.128, -12.541, 23.948, 17.764]
  MoveL 553 to (-960, 150, 50) mm, rotated rx 180 ry 0 rz 90 deg; joints [8.243, -51.44, 80.804, -13.637, 22.5, 19.057]
  MoveL 554 to (-960, 150, -0.5) mm, rotated rx 180 ry 0 rz 90 deg; joints [8.243, -50.087, 81.331, -14.804, 20.677, 20.312]
  MoveL 555 to (-960, 150, 50) mm, rotated rx 180 ry 0 rz 90 deg; joints [8.243, -51.44, 80.804, -13.637, 22.5, 19.057]
  MoveL 556 to (-960, 200, 50) mm, rotated rx 180 ry 0 rz 90 deg; joints [8.444, -53.539, 84.347, -14.844, 21.143, 20.466]
  MoveL 557 to (-960, 200, -0.5) mm, rotated rx 180 ry 0 rz 90 deg; joints [8.444, -52.139, 84.871, -16.245, 19.289, 21.958]
  MoveL 558 to (-960, 200, 50) mm, rotated rx 180 ry 0 rz 90 deg; joints [8.444, -53.539, 84.347, -14.844, 21.143, 20.466]
  MoveL 559 to (-960, 250, 50) mm, rotated rx 180 ry 0 rz 90 deg; joints [8.655, -55.595, 87.772, -16.176, 19.872, 22.005]
  MoveL 560 to (-960, 250, -0.5) mm, rotated rx 180 ry 0 rz 90 deg; joints [8.655, -54.148, 88.296, -17.858, 17.987, 23.784]
  MoveL 561 to (-960, 250, 50) mm, rotated rx 180 ry 0 rz 90 deg; joints [8.655, -55.595, 87.772, -16.176, 19.872, 22.005]
  MoveL 562 to (-960, 300, 50) mm, rotated rx 180 ry 0 rz 90 deg; joints [8.876, -57.618, 91.093, -17.646, 18.684, 23.689]
  MoveL 563 to (-960, 300, -0.5) mm, rotated rx 180 ry 0 rz 90 deg; joints [8.876, -56.121, 91.618, -19.669, 16.768, 25.813]
  MoveL 564 to (-960, 300, 50) mm, rotated rx 180 ry 0 rz 90 deg; joints [8.876, -57.618, 91.093, -17.646, 18.684, 23.689]
  MoveL 565 to (-960, 350, 50) mm, rotated rx 180 ry 0 rz 90 deg; joints [9.11, -59.614, 94.321, -19.265, 17.577, 25.531]
  MoveL 566 to (-960, 350, -0.5) mm, rotated rx 180 ry 0 rz 90 deg; joints [9.11, -58.066, 94.848, -21.701, 15.632, 28.073]
  MoveL 567 to (-960, 350, 50) mm, rotated rx 180 ry 0 rz 90 deg; joints [9.11, -59.614, 94.321, -19.265, 17.577, 25.531]
  MoveL 568 to (-960, 400, 50) mm, rotated rx 180 ry 0 rz 90 deg; joints [9.355, -61.59, 97.464, -21.047, 16.55, 27.543]
  MoveL 569 to (-960, 400, -0.5) mm, rotated rx 180 ry 0 rz 90 deg; joints [9.355, -59.987, 97.995, -23.981, 14.579, 30.588]
  MoveL 570 to (-960, 400, 50) mm, rotated rx 180 ry 0 rz 90 deg; joints [9.355, -61.59, 97.464, -21.047, 16.55, 27.543]
  MoveL 571 to (-960, 450, 50) mm, rotated rx 180 ry 0 rz 90 deg; joints [9.615, -63.552, 100.53, -23.001, 15.605, 29.737]
  MoveL 572 to (-960, 450, -0.5) mm, rotated rx 180 ry 0 rz 90 deg; joints [9.615, -61.893, 101.067, -26.532, 13.61, 33.385]
  MoveL 573 to (-960, 450, 50) mm, rotated rx 180 ry 0 rz 90 deg; joints [9.615, -63.552, 100.53, -23.001, 15.605, 29.737]
  MoveL 574 to (-960, 500, 50) mm, rotated rx -180 ry 0 rz 90 deg; joints [9.889, -65.506, 103.526, -25.133, 14.742, 32.119]
  MoveL 575 to (-960, 500, -0.5) mm, rotated rx 180 ry 0 rz 90 deg; joints [9.889, -63.787, 104.07, -29.374, 12.729, 36.483]
  MoveL 576 to (-960, 500, 50) mm, rotated rx -180 ry 0 rz 90 deg; joints [9.889, -65.506, 103.526, -25.133, 14.742, 32.119]
  MoveL 577 to (-960, 550, 50) mm, rotated rx -180 ry 0 rz 90 deg; joints [10.178, -67.457, 106.457, -27.444, 13.963, 34.69]
  MoveL 578 to (-960, 550, -0.5) mm, rotated rx -180 ry 0 rz 90 deg; joints [10.178, -65.675, 107.01, -32.518, 11.939, 39.896]
  MoveL 579 to (-960, 550, 50) mm, rotated rx -180 ry 0 rz 90 deg; joints [10.178, -67.457, 106.457, -27.444, 13.963, 34.69]
  MoveL 580 to (-960, 600, 50) mm, rotated rx -180 ry 0 rz 90 deg; joints [10.486, -69.411, 109.328, -29.925, 13.272, 37.444]
  MoveL 581 to (-960, 600, -0.5) mm, rotated rx 180 ry 0 rz 90 deg; joints [10.486, -67.563, 109.891, -35.962, 11.246, 43.621]
  MoveL 582 to (-960, 600, 50) mm, rotated rx -180 ry 0 rz 90 deg; joints [10.486, -69.411, 109.328, -29.925, 13.272, 37.444]
  MoveL 583 to (-960, 650, 50) mm, rotated rx 180 ry 0 rz 90 deg; joints [10.812, -71.374, 112.144, -32.557, 12.672, 40.361]
  MoveL 584 to (-960, 650, -0.5) mm, rotated rx -180 ry 0 rz 90 deg; joints [10.812, -69.456, 112.719, -39.682, 10.654, 47.635]
  MoveL 585 to (-960, 650, 50) mm, rotated rx 180 ry 0 rz 90 deg; joints [10.812, -71.374, 112.144, -32.557, 12.672, 40.361]
  MoveL 586 to (-960, 700, 50) mm, rotated rx 180 ry 0 rz 90 deg; joints [11.158, -73.351, 114.908, -35.305, 12.165, 43.409]
  MoveL 587 to (-960, 700, -0.5) mm, rotated rx 180 ry 0 rz 90 deg; joints [11.158, -71.358, 115.496, -43.626, 10.167, 51.888]
  MoveL 588 to (-960, 700, 50) mm, rotated rx 180 ry 0 rz 90 deg; joints [11.158, -73.351, 114.908, -35.305, 12.165, 43.409]
  MoveL 589 to (-960, 750, 50) mm, rotated rx 180 ry 0 rz 90 deg; joints [11.527, -75.35, 117.622, -38.12, 11.755, 46.538]
  MoveL 590 to (-960, 750, -0.5) mm, rotated rx -180 ry 0 rz 90 deg; joints [11.527, -73.277, 118.226, -47.711, 9.788, 56.299]
  MoveL 591 to (-960, 750, 50) mm, rotated rx 180 ry 0 rz 90 deg; joints [11.527, -75.35, 117.622, -38.12, 11.755, 46.538]
  MoveL 592 to (-960, 800, 50) mm, rotated rx -180 ry 0 rz 90 deg; joints [11.922, -77.376, 120.29, -40.935, 11.444, 49.684]
  MoveL 593 to (-960, 800, -0.5) mm, rotated rx -180 ry 0 rz 90 deg; joints [11.922, -75.219, 120.911, -51.824, 9.519, 60.755]
  MoveL 594 to (-960, 800, 50) mm, rotated rx -180 ry 0 rz 90 deg; joints [11.922, -77.376, 120.29, -40.935, 11.444, 49.684]
  MoveL 595 to (-960, 850, 50) mm, rotated rx -180 ry 0 rz 90 deg; joints [12.343, -79.437, 122.914, -43.669, 11.235, 52.767]
  MoveL 596 to (-960, 850, -0.5) mm, rotated rx 180 ry 0 rz 90 deg; joints [12.343, -77.19, 123.555, -55.826, 9.358, 65.12]
  MoveL 597 to (-960, 850, 50) mm, rotated rx -180 ry 0 rz 90 deg; joints [12.343, -79.437, 122.914, -43.669, 11.235, 52.767]
  MoveL 598 to (-960, 900, 50) mm, rotated rx 180 ry 0 rz 90 deg; joints [12.795, -81.542, 125.495, -46.23, 11.128, 55.696]
  MoveL 599 to (-960, 900, -0.5) mm, rotated rx 180 ry 0 rz 90 deg; joints [12.795, -79.197, 126.158, -59.569, 9.302, 69.247]
  MoveL 600 to (-960, 900, 50) mm, rotated rx 180 ry 0 rz 90 deg; joints [12.795, -81.542, 125.495, -46.23, 11.128, 55.696]
  MoveL 601 to (-960, 950, 50) mm, rotated rx 180 ry 0 rz 90 deg; joints [13.281, -83.699, 128.035, -48.524, 11.126, 58.379]
  MoveL 602 to (-960, 950, -0.5) mm, rotated rx 180 ry 0 rz 90 deg; joints [13.281, -81.251, 128.722, -62.907, 9.346, 72.991]
  MoveL 603 to (-960, 950, 50) mm, rotated rx 180 ry 0 rz 90 deg; joints [13.281, -83.699, 128.035, -48.524, 11.126, 58.379]
  MoveL 604 to (-960, 1000, 50) mm, rotated rx -180 ry 0 rz 90 deg; joints [13.805, -85.918, 130.534, -50.459, 11.229, 60.725]
  MoveL 605 to (-960, 1000, -0.5) mm, rotated rx -180 ry 0 rz 90 deg; joints [13.805, -83.36, 131.248, -65.712, 9.483, 76.226]
  MoveL 606 to (-960, 1000, 50) mm, rotated rx -180 ry 0 rz 90 deg; joints [13.805, -85.918, 130.534, -50.459, 11.229, 60.725]
  MoveL 607 to (-960, 1050, 50) mm, rotated rx -180 ry 0 rz 90 deg; joints [14.37, -88.213, 132.993, -51.955, 11.439, 62.657]
  MoveL 608 to (-960, 1050, -0.5) mm, rotated rx 180 ry 0 rz 90 deg; joints [14.37, -85.535, 133.737, -67.878, 9.707, 78.849]
  MoveL 609 to (-960, 1050, 50) mm, rotated rx -180 ry 0 rz 90 deg; joints [14.37, -88.213, 132.993, -51.955, 11.439, 62.657]
  MoveL 610 to (-960, 1100, 50) mm, rotated rx 180 ry 0 rz 90 deg; joints [14.983, -90.597, 135.411, -52.948, 11.763, 64.111]
  MoveL 611 to (-960, 1100, -0.5) mm, rotated rx 180 ry 0 rz 90 deg; joints [14.983, -87.791, 136.19, -69.33, 10.014, 80.787]
  MoveL 612 to (-960, 1100, 50) mm, rotated rx 180 ry 0 rz 90 deg; joints [14.983, -90.597, 135.411, -52.948, 11.763, 64.111]
  MoveL 613 to (-960, 1150, 50) mm, rotated rx 180 ry 0 rz 90 deg; joints [15.649, -93.086, 137.789, -53.393, 12.208, 65.045]
  MoveL 614 to (-960, 1150, -0.5) mm, rotated rx -180 ry 0 rz 90 deg; joints [15.649, -90.143, 138.606, -70.015, 10.407, 81.99]
  MoveL 615 to (-960, 1150, 50) mm, rotated rx 180 ry 0 rz 90 deg; joints [15.649, -93.086, 137.789, -53.393, 12.208, 65.045]
  MoveL 616 to (-960, 1200, 50) mm, rotated rx -180 ry 0 rz 90 deg; joints [16.375, -95.7, 140.124, -53.269, 12.79, 65.44]
  MoveL 617 to (-960, 1200, -0.5) mm, rotated rx -180 ry 0 rz 90 deg; joints [16.375, -92.61, 140.984, -69.906, 10.89, 82.431]
  MoveL 618 to (-960, 1200, 50) mm, rotated rx -180 ry 0 rz 90 deg; joints [16.375, -95.7, 140.124, -53.269, 12.79, 65.44]
  MoveL 619 to (-1030, 50, 50) mm, rotated rx 180 ry 0 rz 90 deg; joints [9.672, -46.589, 72.451, -13.854, 26.203, 20.023]
  MoveL 620 to (-1030, 50, -0.5) mm, rotated rx 180 ry 0 rz 90 deg; joints [9.672, -45.336, 72.993, -14.793, 24.463, 21.061]
  MoveL 621 to (-1030, 50, 50) mm, rotated rx 180 ry 0 rz 90 deg; joints [9.672, -46.589, 72.451, -13.854, 26.203, 20.023]
  MoveL 622 to (-1030, 100, 50) mm, rotated rx 180 ry 0 rz 90 deg; joints [9.896, -48.807, 76.297, -15.014, 24.676, 21.418]
  MoveL 623 to (-1030, 100, -0.5) mm, rotated rx 180 ry 0 rz 90 deg; joints [9.896, -47.509, 76.831, -16.13, 22.911, 22.637]
  MoveL 624 to (-1030, 100, 50) mm, rotated rx 180 ry 0 rz 90 deg; joints [9.896, -48.807, 76.297, -15.014, 24.676, 21.418]
  MoveL 625 to (-1030, 150, 50) mm, rotated rx 180 ry 0 rz 90 deg; joints [10.13, -50.959, 79.986, -16.283, 23.251, 22.927]
  MoveL 626 to (-1030, 150, -0.5) mm, rotated rx 180 ry 0 rz 90 deg; joints [10.13, -49.616, 80.514, -17.609, 21.461, 24.361]
  MoveL 627 to (-1030, 150, 50) mm, rotated rx 180 ry 0 rz 90 deg; joints [10.13, -50.959, 79.986, -16.283, 23.251, 22.927]
  MoveL 628 to (-1030, 200, 50) mm, rotated rx -180 ry 0 rz 90 deg; joints [10.375, -53.057, 83.538, -17.671, 21.923, 24.563]
  MoveL 629 to (-1030, 200, -0.5) mm, rotated rx 180 ry 0 rz 90 deg; joints [10.375, -51.668, 84.063, -19.249, 20.107, 26.253]
  MoveL 630 to (-1030, 200, 50) mm, rotated rx -180 ry 0 rz 90 deg; joints [10.375, -53.057, 83.538, -17.671, 21.923, 24.563]
  MoveL 631 to (-1030, 250, 50) mm, rotated rx -180 ry 0 rz 90 deg; joints [10.632, -55.111, 86.97, -19.191, 20.685, 26.337]
  MoveL 632 to (-1030, 250, -0.5) mm, rotated rx 180 ry 0 rz 90 deg; joints [10.632, -53.675, 87.493, -21.068, 18.845, 28.331]
  MoveL 633 to (-1030, 250, 50) mm, rotated rx -180 ry 0 rz 90 deg; joints [10.632, -55.111, 86.97, -19.191, 20.685, 26.337]
  MoveL 634 to (-1030, 300, 50) mm, rotated rx -180 ry 0 rz 90 deg; joints [10.902, -57.129, 90.294, -20.852, 19.535, 28.261]
  MoveL 635 to (-1030, 300, -0.5) mm, rotated rx -180 ry 0 rz 90 deg; joints [10.902, -55.644, 90.818, -23.085, 17.672, 30.617]
  MoveL 636 to (-1030, 300, 50) mm, rotated rx -180 ry 0 rz 90 deg; joints [10.902, -57.129, 90.294, -20.852, 19.535, 28.261]
  MoveL 637 to (-1030, 350, 50) mm, rotated rx 180 ry 0 rz 90 deg; joints [11.187, -59.118, 93.523, -22.666, 18.471, 30.345]
  MoveL 638 to (-1030, 350, -0.5) mm, rotated rx -180 ry 0 rz 90 deg; joints [11.187, -57.582, 94.049, -25.32, 16.587, 33.129]
  MoveL 639 to (-1030, 350, 50) mm, rotated rx 180 ry 0 rz 90 deg; joints [11.187, -59.118, 93.523, -22.666, 18.471, 30.345]
  MoveL 640 to (-1030, 400, 50) mm, rotated rx -180 ry 0 rz 90 deg; joints [11.486, -61.085, 96.665, -24.638, 17.493, 32.599]
  MoveL 641 to (-1030, 400, -0.5) mm, rotated rx 180 ry 0 rz 90 deg; joints [11.486, -59.496, 97.195, -27.79, 15.592, 35.887]
  MoveL 642 to (-1030, 400, 50) mm, rotated rx -180 ry 0 rz 90 deg; joints [11.486, -61.085, 96.665, -24.638, 17.493, 32.599]
  MoveL 643 to (-1030, 450, 50) mm, rotated rx -180 ry 0 rz 90 deg; joints [11.801, -63.036, 99.728, -26.774, 16.601, 35.028]
  MoveL 644 to (-1030, 450, -0.5) mm, rotated rx 180 ry 0 rz 90 deg; joints [11.801, -61.391, 100.263, -30.505, 14.687, 38.902]
  MoveL 645 to (-1030, 450, 50) mm, rotated rx -180 ry 0 rz 90 deg; joints [11.801, -63.036, 99.728, -26.774, 16.601, 35.028]
  MoveL 646 to (-1030, 500, 50) mm, rotated rx 180 ry 0 rz 90 deg; joints [12.134, -64.976, 102.719, -29.073, 15.797, 37.632]
  MoveL 647 to (-1030, 500, -0.5) mm, rotated rx 180 ry 0 rz 90 deg; joints [12.134, -63.274, 103.261, -33.473, 13.877, 42.182]
  MoveL 648 to (-1030, 500, 50) mm, rotated rx 180 ry 0 rz 90 deg; joints [12.134, -64.976, 102.719, -29.073, 15.797, 37.632]
  MoveL 649 to (-1030, 550, 50) mm, rotated rx 180 ry 0 rz 90 deg; joints [12.486, -66.911, 105.644, -31.527, 15.082, 40.403]
  MoveL 650 to (-1030, 550, -0.5) mm, rotated rx 180 ry 0 rz 90 deg; joints [12.486, -65.148, 106.194, -36.686, 13.164, 45.722]
  MoveL 651 to (-1030, 550, 50) mm, rotated rx 180 ry 0 rz 90 deg; joints [12.486, -66.911, 105.644, -31.527, 15.082, 40.403]
  MoveL 652 to (-1030, 600, 50) mm, rotated rx 180 ry 0 rz 90 deg; joints [12.858, -68.847, 108.507, -34.118, 14.459, 43.326]
  MoveL 653 to (-1030, 600, -0.5) mm, rotated rx 180 ry 0 rz 90 deg; joints [12.858, -67.019, 109.067, -40.123, 12.552, 49.5]
  MoveL 654 to (-1030, 600, 50) mm, rotated rx 180 ry 0 rz 90 deg; joints [12.858, -68.847, 108.507, -34.118, 14.459, 43.326]
  MoveL 655 to (-1030, 650, 50) mm, rotated rx 180 ry 0 rz 90 deg; joints [13.253, -70.789, 111.313, -36.819, 13.93, 46.375]
  MoveL 656 to (-1030, 650, -0.5) mm, rotated rx 180 ry 0 rz 90 deg; joints [13.253, -68.892, 111.884, -43.743, 12.044, 53.479]
  MoveL 657 to (-1030, 650, 50) mm, rotated rx 180 ry 0 rz 90 deg; joints [13.253, -70.789, 111.313, -36.819, 13.93, 46.375]
  MoveL 658 to (-1030, 700, 50) mm, rotated rx 180 ry 0 rz 90 deg; joints [13.673, -72.743, 114.065, -39.59, 13.499, 49.51]
  MoveL 659 to (-1030, 700, -0.5) mm, rotated rx 180 ry 0 rz 90 deg; joints [13.673, -70.773, 114.649, -47.485, 11.643, 57.597]
  MoveL 660 to (-1030, 700, 50) mm, rotated rx 180 ry 0 rz 90 deg; joints [13.673, -72.743, 114.065, -39.59, 13.499, 49.51]
  MoveL 661 to (-1030, 750, 50) mm, rotated rx 180 ry 0 rz 90 deg; joints [14.119, -74.713, 116.766, -42.378, 13.165, 52.68]
  MoveL 662 to (-1030, 750, -0.5) mm, rotated rx 180 ry 0 rz 90 deg; joints [14.119, -72.667, 117.365, -51.267, 11.35, 61.775]
  MoveL 663 to (-1030, 750, 50) mm, rotated rx 180 ry 0 rz 90 deg; joints [14.119, -74.713, 116.766, -42.378, 13.165, 52.68]
  MoveL 664 to (-1030, 800, 50) mm, rotated rx 180 ry 0 rz 90 deg; joints [14.595, -76.707, 119.42, -45.12, 12.932, 55.824]
  MoveL 665 to (-1030, 800, -0.5) mm, rotated rx -180 ry 0 rz 90 deg; joints [14.595, -74.579, 120.035, -54.989, 11.164, 65.913]
  MoveL 666 to (-1030, 800, 50) mm, rotated rx 180 ry 0 rz 90 deg; joints [14.595, -76.707, 119.42, -45.12, 12.932, 55.824]
  MoveL 667 to (-1030, 850, 50) mm, rotated rx 180 ry 0 rz 90 deg; joints [15.104, -78.732, 122.027, -47.744, 12.8, 58.871]
  MoveL 668 to (-1030, 850, -0.5) mm, rotated rx -180 ry 0 rz 90 deg; joints [15.104, -76.516, 122.661, -58.544, 11.083, 69.907]
  MoveL 669 to (-1030, 850, 50) mm, rotated rx 180 ry 0 rz 90 deg; joints [15.104, -78.732, 122.027, -47.744, 12.8, 58.871]
  MoveL 670 to (-1030, 900, 50) mm, rotated rx 180 ry 0 rz 90 deg; joints [15.648, -80.794, 124.59, -50.176, 12.769, 61.749]
  MoveL 671 to (-1030, 900, -0.5) mm, rotated rx -180 ry 0 rz 90 deg; joints [15.648, -78.485, 125.244, -61.821, 11.102, 73.649]
  MoveL 672 to (-1030, 900, 50) mm, rotated rx 180 ry 0 rz 90 deg; joints [15.648, -80.794, 124.59, -50.176, 12.769, 61.749]
  MoveL 673 to (-1030, 950, 50) mm, rotated rx 180 ry 0 rz 90 deg; joints [16.231, -82.902, 127.109, -52.34, 12.838, 64.384]
  MoveL 674 to (-1030, 950, -0.5) mm, rotated rx 180 ry 0 rz 90 deg; joints [16.231, -80.493, 127.787, -64.722, 11.218, 77.041]
  MoveL 675 to (-1030, 950, 50) mm, rotated rx 180 ry 0 rz 90 deg; joints [16.231, -82.902, 127.109, -52.34, 12.838, 64.384]
  MoveL 676 to (-1030, 1000, 50) mm, rotated rx 180 ry 0 rz 90 deg; joints [16.859, -85.064, 129.586, -54.169, 13.01, 66.711]
  MoveL 677 to (-1030, 1000, -0.5) mm, rotated rx 180 ry 0 rz 90 deg; joints [16.859, -82.549, 130.29, -67.161, 11.423, 80]
  MoveL 678 to (-1030, 1000, 50) mm, rotated rx 180 ry 0 rz 90 deg; joints [16.859, -85.064, 129.586, -54.169, 13.01, 66.711]
  MoveL 679 to (-1030, 1050, 50) mm, rotated rx 180 ry 0 rz 90 deg; joints [17.536, -87.292, 132.021, -55.604, 13.285, 68.673]
  MoveL 680 to (-1030, 1050, -0.5) mm, rotated rx 180 ry 0 rz 90 deg; joints [17.536, -84.662, 132.753, -69.071, 11.713, 82.462]
  MoveL 681 to (-1030, 1050, 50) mm, rotated rx 180 ry 0 rz 90 deg; joints [17.536, -87.292, 132.021, -55.604, 13.285, 68.673]
  MoveL 682 to (-1030, 1100, 50) mm, rotated rx 180 ry 0 rz 90 deg; joints [18.267, -89.597, 134.414, -56.6, 13.667, 70.227]
  MoveL 683 to (-1030, 1100, -0.5) mm, rotated rx -180 ry 0 rz 90 deg; joints [18.267, -86.845, 135.178, -70.402, 12.086, 84.38]
  MoveL 684 to (-1030, 1100, 50) mm, rotated rx 180 ry 0 rz 90 deg; joints [18.267, -89.597, 134.414, -56.6, 13.667, 70.227]
  MoveL 685 to (-1030, 1150, 50) mm, rotated rx 180 ry 0 rz 90 deg; joints [19.06, -91.993, 136.763, -57.125, 14.163, 71.343]
  MoveL 686 to (-1030, 1150, -0.5) mm, rotated rx 180 ry 0 rz 90 deg; joints [19.06, -89.111, 137.563, -71.123, 12.544, 85.724]
  MoveL 687 to (-1030, 1150, 50) mm, rotated rx 180 ry 0 rz 90 deg; joints [19.06, -91.993, 136.763, -57.125, 14.163, 71.343]
  MoveL 688 to (-1030, 1200, 50) mm, rotated rx -180 ry 0 rz 90 deg; joints [19.921, -94.496, 139.068, -57.165, 14.785, 72.009]
  MoveL 689 to (-1030, 1200, -0.5) mm, rotated rx -180 ry 0 rz 90 deg; joints [19.921, -91.474, 139.908, -71.214, 13.091, 86.478]
  MoveL 690 to (-1030, 1200, 50) mm, rotated rx -180 ry 0 rz 90 deg; joints [19.921, -94.496, 139.068, -57.165, 14.785, 72.009]
  MoveL 691 to (-1100, 50, 50) mm, rotated rx -180 ry 0 rz 90 deg; joints [11.457, -45.999, 71.42, -15.959, 27.043, 23.24]
  MoveL 692 to (-1100, 50, -0.5) mm, rotated rx 180 ry 0 rz 90 deg; joints [11.457, -44.757, 71.966, -16.99, 25.329, 24.389]
  MoveL 693 to (-1100, 50, 50) mm, rotated rx -180 ry 0 rz 90 deg; joints [11.457, -45.999, 71.42, -15.959, 27.043, 23.24]
  MoveL 694 to (-1100, 100, 50) mm, rotated rx 180 ry 0 rz 90 deg; joints [11.72, -48.223, 75.288, -17.251, 25.534, 24.811]
  MoveL 695 to (-1100, 100, -0.5) mm, rotated rx 180 ry 0 rz 90 deg; joints [11.72, -46.937, 75.824, -18.468, 23.8, 26.15]
  MoveL 696 to (-1100, 100, 50) mm, rotated rx 180 ry 0 rz 90 deg; joints [11.72, -48.223, 75.288, -17.251, 25.534, 24.811]
  MoveL 697 to (-1100, 150, 50) mm, rotated rx 180 ry 0 rz 90 deg; joints [11.995, -50.377, 78.994, -18.655, 24.134, 26.5]
  MoveL 698 to (-1100, 150, -0.5) mm, rotated rx 180 ry 0 rz 90 deg; joints [11.995, -49.047, 79.523, -20.091, 22.379, 28.063]
  MoveL 699 to (-1100, 150, 50) mm, rotated rx 180 ry 0 rz 90 deg; joints [11.995, -50.377, 78.994, -18.655, 24.134, 26.5]
  MoveL 700 to (-1100, 200, 50) mm, rotated rx -180 ry 0 rz 90 deg; joints [12.283, -52.475, 82.558, -20.181, 22.834, 28.317]
  MoveL 701 to (-1100, 200, -0.5) mm, rotated rx 180 ry 0 rz 90 deg; joints [12.283, -51.1, 83.083, -21.874, 21.059, 30.143]
  MoveL 702 to (-1100, 200, 50) mm, rotated rx -180 ry 0 rz 90 deg; joints [12.283, -52.475, 82.558, -20.181, 22.834, 28.317]
  MoveL 703 to (-1100, 250, 50) mm, rotated rx 180 ry 0 rz 90 deg; joints [12.585, -54.526, 85.997, -21.837, 21.631, 30.273]
  MoveL 704 to (-1100, 250, -0.5) mm, rotated rx 180 ry 0 rz 90 deg; joints [12.585, -53.104, 86.521, -23.832, 19.837, 32.406]
  MoveL 705 to (-1100, 250, 50) mm, rotated rx 180 ry 0 rz 90 deg; joints [12.585, -54.526, 85.997, -21.837, 21.631, 30.273]
  MoveL 706 to (-1100, 300, 50) mm, rotated rx -180 ry 0 rz 90 deg; joints [12.901, -56.539, 89.327, -23.632, 20.519, 32.377]
  MoveL 707 to (-1100, 300, -0.5) mm, rotated rx -180 ry 0 rz 90 deg; joints [12.901, -55.068, 89.851, -25.98, 18.709, 34.869]
  MoveL 708 to (-1100, 300, 50) mm, rotated rx -180 ry 0 rz 90 deg; joints [12.901, -56.539, 89.327, -23.632, 20.519, 32.377]
  MoveL 709 to (-1100, 350, 50) mm, rotated rx -180 ry 0 rz 90 deg; joints [13.234, -58.52, 92.558, -25.571, 19.499, 34.635]
  MoveL 710 to (-1100, 350, -0.5) mm, rotated rx 180 ry 0 rz 90 deg; joints [13.234, -57, 93.083, -28.328, 17.675, 37.543]
  MoveL 711 to (-1100, 350, 50) mm, rotated rx -180 ry 0 rz 90 deg; joints [13.234, -58.52, 92.558, -25.571, 19.499, 34.635]
  MoveL 712 to (-1100, 400, 50) mm, rotated rx 180 ry 0 rz 90 deg; joints [13.584, -60.477, 95.699, -27.657, 18.569, 37.052]
  MoveL 713 to (-1100, 400, -0.5) mm, rotated rx -180 ry 0 rz 90 deg; joints [13.584, -58.905, 96.228, -30.885, 16.735, 40.439]
  MoveL 714 to (-1100, 400, 50) mm, rotated rx 180 ry 0 rz 90 deg; joints [13.584, -60.477, 95.699, -27.657, 18.569, 37.052]
  MoveL 715 to (-1100, 450, 50) mm, rotated rx 180 ry 0 rz 90 deg; joints [13.953, -62.415, 98.76, -29.889, 17.729, 39.628]
  MoveL 716 to (-1100, 450, -0.5) mm, rotated rx 180 ry 0 rz 90 deg; joints [13.953, -60.789, 99.293, -33.654, 15.892, 43.56]
  MoveL 717 to (-1100, 450, 50) mm, rotated rx 180 ry 0 rz 90 deg; joints [13.953, -62.415, 98.76, -29.889, 17.729, 39.628]
  MoveL 718 to (-1100, 500, 50) mm, rotated rx 180 ry 0 rz 90 deg; joints [14.342, -64.341, 101.746, -32.26, 16.981, 42.357]
  MoveL 719 to (-1100, 500, -0.5) mm, rotated rx 180 ry 0 rz 90 deg; joints [14.342, -62.658, 102.285, -36.628, 15.146, 46.901]
  MoveL 720 to (-1100, 500, 50) mm, rotated rx 180 ry 0 rz 90 deg; joints [14.342, -64.341, 101.746, -32.26, 16.981, 42.357]
  MoveL 721 to (-1100, 550, 50) mm, rotated rx -180 ry 0 rz 90 deg; joints [14.752, -66.258, 104.663, -34.757, 16.326, 45.226]
  MoveL 722 to (-1100, 550, -0.5) mm, rotated rx 180 ry 0 rz 90 deg; joints [14.752, -64.516, 105.211, -39.789, 14.502, 50.445]
  MoveL 723 to (-1100, 550, 50) mm, rotated rx -180 ry 0 rz 90 deg; joints [14.752, -66.258, 104.663, -34.757, 16.326, 45.226]
  MoveL 724 to (-1100, 600, 50) mm, rotated rx -180 ry 0 rz 90 deg; joints [15.187, -68.173, 107.517, -37.357, 15.766, 48.215]
  MoveL 725 to (-1100, 600, -0.5) mm, rotated rx 180 ry 0 rz 90 deg; joints [15.187, -66.368, 108.074, -43.108, 13.96, 54.164]
  MoveL 726 to (-1100, 600, 50) mm, rotated rx -180 ry 0 rz 90 deg; joints [15.187, -68.173, 107.517, -37.357, 15.766, 48.215]
  MoveL 727 to (-1100, 650, 50) mm, rotated rx -180 ry 0 rz 90 deg; joints [15.647, -70.091, 110.312, -40.027, 15.302, 51.292]
  MoveL 728 to (-1100, 650, -0.5) mm, rotated rx -180 ry 0 rz 90 deg; joints [15.647, -68.219, 110.879, -46.538, 13.524, 58.013]
  MoveL 729 to (-1100, 650, 50) mm, rotated rx -180 ry 0 rz 90 deg; joints [15.647, -70.091, 110.312, -40.027, 15.302, 51.292]
  MoveL 730 to (-1100, 700, 50) mm, rotated rx 180 ry 0 rz 90 deg; joints [16.135, -72.017, 113.051, -42.729, 14.936, 54.419]
  MoveL 731 to (-1100, 700, -0.5) mm, rotated rx 180 ry 0 rz 90 deg; joints [16.135, -70.075, 113.63, -50.019, 13.193, 61.933]
  MoveL 732 to (-1100, 700, 50) mm, rotated rx 180 ry 0 rz 90 deg; joints [16.135, -72.017, 113.051, -42.729, 14.936, 54.419]
  MoveL 733 to (-1100, 750, 50) mm, rotated rx -180 ry 0 rz 90 deg; joints [16.653, -73.956, 115.738, -45.41, 14.67, 57.548]
  MoveL 734 to (-1100, 750, -0.5) mm, rotated rx 180 ry 0 rz 90 deg; joints [16.653, -71.94, 116.331, -53.478, 12.969, 65.854]
  MoveL 735 to (-1100, 750, 50) mm, rotated rx -180 ry 0 rz 90 deg; joints [16.653, -73.956, 115.738, -45.41, 14.67, 57.548]
  MoveL 736 to (-1100, 800, 50) mm, rotated rx 180 ry 0 rz 90 deg; joints [17.205, -75.914, 118.374, -48.017, 14.503, 60.624]
  MoveL 737 to (-1100, 800, -0.5) mm, rotated rx 180 ry 0 rz 90 deg; joints [17.205, -73.819, 118.982, -56.834, 12.849, 69.696]
  MoveL 738 to (-1100, 800, 50) mm, rotated rx 180 ry 0 rz 90 deg; joints [17.205, -75.914, 118.374, -48.017, 14.503, 60.624]
  MoveL 739 to (-1100, 850, 50) mm, rotated rx 180 ry 0 rz 90 deg; joints [17.794, -77.897, 120.962, -50.488, 14.435, 63.589]
  MoveL 740 to (-1100, 850, -0.5) mm, rotated rx -180 ry 0 rz 90 deg; joints [17.794, -75.717, 121.588, -60.005, 12.83, 73.379]
  MoveL 741 to (-1100, 850, 50) mm, rotated rx 180 ry 0 rz 90 deg; joints [17.794, -77.897, 120.962, -50.488, 14.435, 63.589]
  MoveL 742 to (-1100, 900, 50) mm, rotated rx 180 ry 0 rz 90 deg; joints [18.423, -79.911, 123.504, -52.764, 14.466, 66.385]
  MoveL 743 to (-1100, 900, -0.5) mm, rotated rx -180 ry 0 rz 90 deg; joints [18.423, -77.642, 124.149, -62.909, 12.908, 76.823]
  MoveL 744 to (-1100, 900, 50) mm, rotated rx 180 ry 0 rz 90 deg; joints [18.423, -79.911, 123.504, -52.764, 14.466, 66.385]
  MoveL 745 to (-1100, 950, 50) mm, rotated rx 180 ry 0 rz 90 deg; joints [19.096, -81.963, 126, -54.788, 14.595, 68.956]
  MoveL 746 to (-1100, 950, -0.5) mm, rotated rx 180 ry 0 rz 90 deg; joints [19.096, -79.599, 126.667, -65.477, 13.079, 79.962]
  MoveL 747 to (-1100, 950, 50) mm, rotated rx 180 ry 0 rz 90 deg; joints [19.096, -81.963, 126, -54.788, 14.595, 68.956]
  MoveL 748 to (-1100, 1000, 50) mm, rotated rx -180 ry 0 rz 90 deg; joints [19.818, -84.062, 128.452, -56.507, 14.823, 71.255]
  MoveL 749 to (-1100, 1000, -0.5) mm, rotated rx 180 ry 0 rz 90 deg; joints [19.818, -81.596, 129.143, -67.648, 13.338, 82.737]
  MoveL 750 to (-1100, 1000, 50) mm, rotated rx -180 ry 0 rz 90 deg; joints [19.818, -84.062, 128.452, -56.507, 14.823, 71.255]
  MoveL 751 to (-1100, 1050, 50) mm, rotated rx -180 ry 0 rz 90 deg; joints [20.595, -86.215, 130.859, -57.88, 15.151, 73.24]
  MoveL 752 to (-1100, 1050, -0.5) mm, rotated rx 180 ry 0 rz 90 deg; joints [20.595, -83.641, 131.577, -69.376, 13.681, 85.106]
  MoveL 753 to (-1100, 1050, 50) mm, rotated rx -180 ry 0 rz 90 deg; joints [20.595, -86.215, 130.859, -57.88, 15.151, 73.24]
  MoveL 754 to (-1100, 1100, 50) mm, rotated rx 180 ry 0 rz 90 deg; joints [21.431, -88.434, 133.222, -58.874, 15.582, 74.881]
  MoveL 755 to (-1100, 1100, -0.5) mm, rotated rx 180 ry 0 rz 90 deg; joints [21.431, -85.744, 133.97, -70.628, 14.108, 87.037]
  MoveL 756 to (-1100, 1100, 50) mm, rotated rx 180 ry 0 rz 90 deg; joints [21.431, -88.434, 133.222, -58.874, 15.582, 74.881]
  MoveL 757 to (-1100, 1150, 50) mm, rotated rx -180 ry 0 rz 90 deg; joints [22.335, -90.728, 135.54, -59.466, 16.121, 76.158]
  MoveL 758 to (-1100, 1150, -0.5) mm, rotated rx 180 ry 0 rz 90 deg; joints [22.335, -87.915, 136.32, -71.381, 14.618, 88.511]
  MoveL 759 to (-1100, 1150, 50) mm, rotated rx -180 ry 0 rz 90 deg; joints [22.335, -90.728, 135.54, -59.466, 16.121, 76.158]
  MoveL 760 to (-1100, 1200, 50) mm, rotated rx -180 ry 0 rz 90 deg; joints [23.315, -93.11, 137.811, -59.644, 16.777, 77.063]
  MoveL 761 to (-1100, 1200, -0.5) mm, rotated rx 180 ry 0 rz 90 deg; joints [23.315, -90.166, 138.628, -71.624, 15.216, 89.521]
  MoveL 762 to (-1100, 1200, 50) mm, rotated rx -180 ry 0 rz 90 deg; joints [23.315, -93.11, 137.811, -59.644, 16.777, 77.063]
  MoveL 763 to (-1170, 50, 50) mm, rotated rx 180 ry 0 rz 90 deg; joints [13.22, -45.305, 70.203, -17.848, 28.007, 26.216]
  MoveL 764 to (-1170, 50, -0.5) mm, rotated rx 180 ry 0 rz 90 deg; joints [13.22, -44.076, 70.752, -18.941, 26.32, 27.444]
  MoveL 765 to (-1170, 50, 50) mm, rotated rx 180 ry 0 rz 90 deg; joints [13.22, -45.305, 70.203, -17.848, 28.007, 26.216]
  MoveL 766 to (-1170, 100, 50) mm, rotated rx 180 ry 0 rz 90 deg; joints [13.521, -47.536, 74.099, -19.242, 26.516, 27.931]
  MoveL 767 to (-1170, 100, -0.5) mm, rotated rx -180 ry 0 rz 90 deg; joints [13.521, -46.264, 74.637, -20.524, 24.813, 29.353]
  MoveL 768 to (-1170, 100, 50) mm, rotated rx 180 ry 0 rz 90 deg; joints [13.521, -47.536, 74.099, -19.242, 26.516, 27.931]
  MoveL 769 to (-1170, 150, 50) mm, rotated rx -180 ry 0 rz 90 deg; joints [13.835, -49.695, 77.825, -20.747, 25.138, 29.763]
  MoveL 770 to (-1170, 150, -0.5) mm, rotated rx 180 ry 0 rz 90 deg; joints [13.835, -48.379, 78.356, -22.248, 23.419, 31.41]
  MoveL 771 to (-1170, 150, 50) mm, rotated rx -180 ry 0 rz 90 deg; joints [13.835, -49.695, 77.825, -20.747, 25.138, 29.763]
